C05558=1105.654,-74.562,-48.566,179.834,5.090,148.924
C05559=1105.648,-74.312,-48.578,179.834,5.095,148.925
C05560=1105.644,-74.063,-48.589,179.834,5.100,148.926
C05561=1105.639,-73.813,-48.600,179.834,5.105,148.927
C05562=1105.634,-73.563,-48.612,179.834,5.110,148.929
C05563=1105.629,-73.349,-48.622,179.834,5.114,148.929
C05564=1105.625,-73.135,-48.631,179.834,5.119,148.931
C05565=1105.620,-72.920,-48.641,179.833,5.123,148.932
C05566=1105.616,-72.706,-48.651,179.834,5.128,148.932
C05567=1105.611,-72.491,-48.660,179.833,5.132,148.933
C05568=1105.607,-72.276,-48.670,179.834,5.137,148.934
C05569=1105.602,-72.063,-48.679,179.833,5.141,148.936
C05570=1105.598,-71.848,-48.689,179.833,5.146,148.936
C05571=1105.593,-71.598,-48.701,179.833,5.151,148.938
C05572=1105.587,-71.349,-48.712,179.833,5.156,148.939
C05573=1105.582,-71.099,-48.724,179.834,5.161,148.940
C05574=1105.577,-70.849,-48.735,179.833,5.166,148.941
C05575=1105.571,-70.599,-48.747,179.833,5.171,148.942
C05576=1105.566,-70.350,-48.757,179.833,5.176,148.943
C05577=1105.561,-70.100,-48.769,179.833,5.181,148.944
C05578=1105.556,-69.850,-48.781,179.833,5.187,148.946
C05579=1105.551,-69.600,-48.793,179.833,5.191,148.947
C05580=1105.546,-69.351,-48.804,179.833,5.196,148.948
C05581=1105.540,-69.101,-48.816,179.833,5.202,148.949
C05582=1105.535,-68.852,-48.827,179.833,5.207,148.950
C05583=1105.530,-68.602,-48.839,179.833,5.212,148.951
C05584=1105.525,-68.352,-48.850,179.833,5.217,148.952
C05585=1105.520,-68.102,-48.862,179.833,5.222,148.953
C05586=1105.515,-67.853,-48.873,179.833,5.227,148.954
C05587=1105.509,-67.603,-48.885,179.833,5.232,148.956
C05588=1105.504,-67.354,-48.896,179.833,5.237,148.957
C05589=1105.499,-67.104,-48.908,179.833,5.242,148.958
C05590=1105.493,-66.854,-48.920,179.833,5.247,148.959
C05591=1105.489,-66.604,-48.931,179.833,5.252,148.960
C05592=1105.483,-66.354,-48.943,179.833,5.257,148.961
C05593=1105.479,-66.105,-48.954,179.833,5.262,148.962
C05594=1105.473,-65.855,-48.966,179.833,5.267,148.963
C05595=1105.468,-65.607,-48.978,179.833,5.272,148.964
C05596=1105.463,-65.357,-48.989,179.833,5.277,148.965
C05597=1105.457,-65.107,-49.001,179.833,5.282,148.966
C05598=1105.453,-64.857,-49.013,179.834,5.288,148.967
C05599=1105.447,-64.607,-49.024,179.834,5.293,148.969
C05600=1105.442,-64.358,-49.036,179.834,5.298,148.970
C05601=1105.437,-64.108,-49.048,179.834,5.303,148.971
C05602=1105.432,-63.858,-49.060,179.834,5.308,148.972
C05603=1105.427,-63.609,-49.072,179.834,5.313,148.973
C05604=1105.422,-63.359,-49.083,179.835,5.317,148.974
C05605=1105.416,-63.109,-49.095,179.835,5.323,148.975
C05606=1105.411,-62.860,-49.106,179.835,5.327,148.976
C05607=1105.406,-62.610,-49.118,179.835,5.332,148.977
C05608=1105.400,-62.361,-49.131,179.835,5.337,148.978
C05609=1105.396,-62.111,-49.142,179.835,5.342,148.979
C05610=1105.390,-61.861,-49.154,179.836,5.347,148.980
C05611=1105.385,-61.611,-49.166,179.835,5.352,148.981
C05612=1105.380,-61.361,-49.177,179.836,5.357,148.982
C05613=1105.375,-61.112,-49.190,179.836,5.362,148.983
C05614=1105.370,-60.862,-49.202,179.836,5.367,148.984
C05615=1105.364,-60.612,-49.213,179.837,5.372,148.985
C05616=1105.360,-60.363,-49.225,179.836,5.377,148.986
C05617=1105.354,-60.113,-49.237,179.837,5.381,148.987
C05618=1105.349,-59.863,-49.249,179.837,5.386,148.988
C05619=1105.345,-59.649,-49.260,179.837,5.390,148.989
C05620=1105.340,-59.435,-49.270,179.837,5.395,148.990
C05621=1105.336,-59.221,-49.280,179.837,5.399,148.991
C05622=1105.332,-59.006,-49.290,179.837,5.403,148.992
C05623=1105.327,-58.792,-49.301,179.837,5.407,148.993
C05624=1105.323,-58.578,-49.311,179.837,5.411,148.994
C05625=1105.319,-58.363,-49.321,179.836,5.415,148.995
C05626=1105.314,-58.148,-49.331,179.836,5.419,148.996
C05627=1105.309,-57.898,-49.343,179.837,5.423,148.997
C05628=1105.304,-57.649,-49.356,179.837,5.428,148.998
C05629=1105.298,-57.399,-49.368,179.836,5.432,148.999
C05630=1105.294,-57.150,-49.380,179.836,5.437,149.000
C05631=1105.289,-56.900,-49.392,179.836,5.443,149.001
C05632=1105.283,-56.650,-49.404,179.836,5.447,149.002
C05633=1105.278,-56.401,-49.416,179.836,5.452,149.003
C05634=1105.273,-56.151,-49.428,179.836,5.456,149.004
C05635=1105.268,-55.902,-49.440,179.836,5.461,149.005
C05636=1105.263,-55.652,-49.452,179.835,5.466,149.006
C05637=1105.257,-55.402,-49.464,179.836,5.471,149.007
C05638=1105.252,-55.153,-49.476,179.835,5.475,149.008
C05639=1105.247,-54.903,-49.488,179.835,5.480,149.009
C05640=1105.242,-54.654,-49.501,179.835,5.485,149.010
C05641=1105.236,-54.404,-49.513,179.835,5.489,149.012
C05642=1105.232,-54.155,-49.525,179.835,5.494,149.012
C05643=1105.226,-53.905,-49.537,179.835,5.499,149.014
C05644=1105.221,-53.655,-49.549,179.834,5.503,149.015
C05645=1105.216,-53.406,-49.561,179.835,5.508,149.016
C05646=1105.211,-53.156,-49.574,179.835,5.513,149.017
C05647=1105.206,-52.906,-49.586,179.834,5.518,149.018
C05648=1105.201,-52.656,-49.599,179.834,5.522,149.019
C05649=1105.195,-52.406,-49.611,179.834,5.527,149.020
C05650=1105.190,-52.157,-49.623,179.834,5.532,149.021
C05651=1105.185,-51.907,-49.635,179.834,5.536,149.022
C05652=1105.180,-51.658,-49.647,179.834,5.542,149.023
C05653=1105.175,-51.408,-49.659,179.833,5.546,149.024
C05654=1105.170,-51.159,-49.671,179.834,5.551,149.025
C05655=1105.165,-50.909,-49.684,179.834,5.556,149.027
C05656=1105.160,-50.659,-49.696,179.833,5.560,149.028
C05657=1105.155,-50.410,-49.709,179.833,5.565,149.029
C05658=1105.149,-50.160,-49.721,179.833,5.569,149.030
C05659=1105.144,-49.910,-49.733,179.833,5.574,149.031
C05660=1105.139,-49.661,-49.746,179.833,5.579,149.032
C05661=1105.134,-49.411,-49.758,179.832,5.583,149.033
C05662=1105.129,-49.162,-49.771,179.832,5.588,149.034
C05663=1105.123,-48.912,-49.782,179.832,5.594,149.035
C05664=1105.119,-48.662,-49.795,179.832,5.598,149.036
C05665=1105.113,-48.412,-49.808,179.832,5.603,149.037
C05666=1105.108,-48.162,-49.820,179.832,5.608,149.039
C05667=1105.103,-47.913,-49.832,179.832,5.612,149.039
C05668=1105.098,-47.664,-49.845,179.832,5.617,149.041
C05669=1105.092,-47.414,-49.857,179.832,5.622,149.042
C05670=1105.088,-47.164,-49.870,179.832,5.626,149.043
C05671=1105.083,-46.915,-49.882,179.831,5.631,149.044
C05672=1105.077,-46.665,-49.894,179.831,5.635,149.045
C05673=1105.072,-46.415,-49.907,179.831,5.640,149.046
C05674=1105.067,-46.166,-49.920,179.831,5.645,149.047
C05675=1105.062,-45.951,-49.931,179.831,5.649,149.048
C05676=1105.058,-45.737,-49.942,179.831,5.653,149.049
C05677=1105.054,-45.523,-49.952,179.830,5.657,149.050
C05678=1105.049,-45.309,-49.963,179.830,5.661,149.051
C05679=1105.044,-45.094,-49.973,179.830,5.665,149.052
C05680=1105.040,-44.880,-49.984,179.830,5.669,149.053
C05681=1105.036,-44.666,-49.995,179.829,5.673,149.054
C05682=1105.032,-44.451,-50.006,179.830,5.678,149.055
C05683=1105.027,-44.202,-50.019,179.829,5.682,149.056
C05684=1105.021,-43.953,-50.031,179.830,5.687,149.057
C05685=1105.016,-43.703,-50.043,179.829,5.691,149.058
C05686=1105.011,-43.453,-50.056,179.829,5.696,149.059
C05687=1105.006,-43.203,-50.069,179.829,5.702,149.060
C05688=1105.001,-42.954,-50.081,179.829,5.705,149.061
C05689=1104.996,-42.705,-50.094,179.829,5.711,149.062
C05690=1104.991,-42.454,-50.107,179.829,5.715,149.063
C05691=1104.985,-42.204,-50.119,179.829,5.720,149.064
C05692=1104.980,-41.955,-50.132,179.829,5.725,149.065
C05693=1104.975,-41.706,-50.145,179.829,5.730,149.066
C05694=1104.971,-41.456,-50.158,179.830,5.735,149.067
C05695=1104.965,-41.206,-50.170,179.830,5.740,149.068
C05696=1104.960,-40.957,-50.183,179.830,5.745,149.069
C05697=1104.955,-40.708,-50.196,179.831,5.750,149.070
C05698=1104.950,-40.457,-50.208,179.831,5.754,149.071
C05699=1104.945,-40.208,-50.221,179.831,5.758,149.072
C05700=1104.939,-39.958,-50.233,179.831,5.763,149.073
C05701=1104.934,-39.709,-50.247,179.831,5.768,149.074
C05702=1104.929,-39.459,-50.260,179.832,5.773,149.075
C05703=1104.924,-39.209,-50.272,179.832,5.778,149.076
C05704=1104.919,-38.960,-50.285,179.833,5.782,149.077
C05705=1104.914,-38.710,-50.298,179.833,5.786,149.078
C05706=1104.908,-38.460,-50.311,179.833,5.791,149.079
C05707=1104.903,-38.211,-50.323,179.833,5.796,149.080
C05708=1104.898,-37.962,-50.336,179.834,5.800,149.080
C05709=1104.894,-37.712,-50.349,179.834,5.804,149.081
C05710=1104.888,-37.462,-50.362,179.834,5.809,149.082
C05711=1104.883,-37.213,-50.375,179.835,5.814,149.083
C05712=1104.878,-36.963,-50.388,179.835,5.819,149.084
C05713=1104.873,-36.713,-50.400,179.835,5.823,149.085
C05714=1104.867,-36.464,-50.414,179.835,5.827,149.086
C05715=1104.863,-36.214,-50.427,179.836,5.832,149.087
C05716=1104.858,-35.964,-50.439,179.836,5.837,149.088
C05717=1104.852,-35.715,-50.452,179.836,5.841,149.089
C05718=1104.847,-35.465,-50.465,179.837,5.845,149.090
C05719=1104.842,-35.215,-50.478,179.837,5.850,149.090
C05720=1104.836,-34.966,-50.491,179.837,5.855,149.091
C05721=1104.832,-34.716,-50.505,179.837,5.859,149.092
C05722=1104.827,-34.467,-50.517,179.838,5.864,149.093
C05723=1104.822,-34.217,-50.531,179.838,5.868,149.094
C05724=1104.816,-33.967,-50.544,179.838,5.872,149.095
C05725=1104.811,-33.718,-50.556,179.838,5.877,149.096
C05726=1104.806,-33.468,-50.570,179.839,5.881,149.097
C05727=1104.801,-33.219,-50.582,179.839,5.885,149.098
C05728=1104.797,-32.969,-50.596,179.840,5.890,149.098
C05729=1104.791,-32.719,-50.609,179.840,5.895,149.099
C05730=1104.786,-32.470,-50.622,179.841,5.899,149.100
C05731=1104.781,-32.256,-50.633,179.841,5.903,149.101
C05732=1104.777,-32.041,-50.644,179.841,5.907,149.102
C05733=1104.772,-31.827,-50.656,179.841,5.910,149.103
C05734=1104.768,-31.613,-50.667,179.842,5.914,149.103
C05735=1104.764,-31.399,-50.678,179.841,5.918,149.104
C05736=1104.760,-31.185,-50.689,179.842,5.921,149.105
C05737=1104.755,-30.970,-50.701,179.843,5.926,149.105
C05738=1104.750,-30.756,-50.712,179.843,5.930,149.106
C05739=1104.746,-30.507,-50.725,179.842,5.934,149.107
C05740=1104.741,-30.257,-50.738,179.843,5.938,149.108
C05741=1104.735,-30.008,-50.751,179.843,5.943,149.109
C05742=1104.731,-29.758,-50.765,179.843,5.947,149.110
C05743=1104.725,-29.509,-50.778,179.844,5.952,149.111
C05744=1104.721,-29.259,-50.791,179.844,5.957,149.112
C05745=1104.715,-29.009,-50.805,179.845,5.961,149.113
C05746=1104.710,-28.760,-50.818,179.844,5.965,149.114
C05747=1104.705,-28.510,-50.831,179.845,5.970,149.115
C05748=1104.700,-28.260,-50.844,179.845,5.975,149.115
C05749=1104.695,-28.011,-50.858,179.845,5.979,149.116
C05750=1104.690,-27.761,-50.871,179.846,5.983,149.117
C05751=1104.685,-27.512,-50.884,179.846,5.988,149.118
C05752=1104.679,-27.263,-50.898,179.847,5.993,149.119
C05753=1104.675,-27.013,-50.911,179.847,5.997,149.120
C05754=1104.669,-26.763,-50.924,179.847,6.002,149.121
C05755=1104.665,-26.513,-50.938,179.847,6.007,149.122
C05756=1104.659,-26.263,-50.951,179.847,6.010,149.123
C05757=1104.655,-26.014,-50.964,179.847,6.015,149.124
C05758=1104.649,-25.764,-50.978,179.847,6.020,149.125
C05759=1104.644,-25.514,-50.991,179.848,6.025,149.126
C05760=1104.639,-25.265,-51.005,179.848,6.030,149.127
C05761=1104.633,-25.015,-51.018,179.848,6.034,149.128
C05762=1104.629,-24.766,-51.032,179.848,6.039,149.129
C05763=1104.623,-24.516,-51.045,179.849,6.044,149.130
C05764=1104.619,-24.267,-51.059,179.849,6.048,149.131
C05765=1104.613,-24.017,-51.072,179.850,6.053,149.132
C05766=1104.608,-23.768,-51.086,179.850,6.058,149.132
C05767=1104.603,-23.518,-51.099,179.849,6.062,149.134
C05768=1104.598,-23.269,-51.113,179.850,6.067,149.135
C05769=1104.593,-23.019,-51.126,179.850,6.071,149.135
C05770=1104.588,-22.770,-51.140,179.851,6.076,149.136
C05771=1104.582,-22.520,-51.153,179.851,6.081,149.137
C05772=1104.578,-22.271,-51.167,179.852,6.086,149.138
C05773=1104.573,-22.020,-51.180,179.852,6.090,149.139
C05774=1104.567,-21.771,-51.194,179.852,6.094,149.140
C05775=1104.563,-21.521,-51.207,179.852,6.099,149.141
C05776=1104.557,-21.272,-51.221,179.853,6.104,149.142
C05777=1104.553,-21.022,-51.234,179.853,6.109,149.143
C05778=1104.547,-20.773,-51.248,179.853,6.113,149.144
C05779=1104.542,-20.524,-51.262,179.853,6.118,149.145
C05780=1104.538,-20.273,-51.275,179.854,6.122,149.146
C05781=1104.532,-20.024,-51.289,179.854,6.127,149.146
C05782=1104.527,-19.774,-51.303,179.855,6.132,149.147
C05783=1104.521,-19.525,-51.317,179.855,6.136,149.148
C05784=1104.517,-19.276,-51.330,179.855,6.140,149.149
C05785=1104.512,-19.025,-51.344,179.856,6.145,149.150
C05786=1104.506,-18.776,-51.358,179.856,6.150,149.151
C05787=1104.503,-18.563,-51.369,179.857,6.153,149.152
C05788=1104.498,-18.348,-51.381,179.857,6.157,149.153
C05789=1104.494,-18.134,-51.393,179.857,6.162,149.153
C05790=1104.489,-17.920,-51.405,179.857,6.166,149.154
C05791=1104.485,-17.706,-51.417,179.858,6.169,149.155
C05792=1104.480,-17.491,-51.428,179.858,6.174,149.156
C05793=1104.476,-17.277,-51.440,179.859,6.177,149.156
C05794=1104.472,-17.064,-51.452,179.859,6.181,149.157
C05795=1104.467,-16.814,-51.466,179.859,6.186,149.158
C05796=1104.462,-16.564,-51.480,179.860,6.190,149.159
C05797=1104.456,-16.315,-51.494,179.860,6.195,149.160
C05798=1104.452,-16.065,-51.507,179.860,6.199,149.161
C05799=1104.447,-15.815,-51.521,179.861,6.204,149.162
C05800=1104.441,-15.566,-51.535,179.861,6.208,149.162
C05801=1104.436,-15.316,-51.549,179.862,6.213,149.163
C05802=1104.431,-15.066,-51.563,179.862,6.218,149.164
C05803=1104.426,-14.818,-51.577,179.862,6.222,149.165
C05804=1104.422,-14.568,-51.591,179.863,6.226,149.166
C05805=1104.416,-14.318,-51.604,179.864,6.231,149.167
C05806=1104.411,-14.069,-51.618,179.864,6.236,149.168
C05807=1104.406,-13.819,-51.633,179.865,6.240,149.169
C05808=1104.401,-13.569,-51.647,179.865,6.245,149.169
C05809=1104.397,-13.320,-51.661,179.865,6.249,149.170
C05810=1104.391,-13.071,-51.674,179.866,6.254,149.171
C05811=1104.386,-12.821,-51.689,179.867,6.258,149.172
C05812=1104.381,-12.571,-51.702,179.867,6.263,149.173
C05813=1104.376,-12.321,-51.717,179.868,6.267,149.174
C05814=1104.370,-12.072,-51.730,179.868,6.272,149.175
C05815=1104.365,-11.822,-51.745,179.868,6.276,149.176
C05816=1104.361,-11.573,-51.758,179.868,6.281,149.176
C05817=1104.356,-11.323,-51.773,179.869,6.285,149.177
C05818=1104.351,-11.074,-51.787,179.870,6.290,149.178
C05819=1104.346,-10.825,-51.801,179.870,6.295,149.179
C05820=1104.341,-10.575,-51.815,179.871,6.299,149.180
C05821=1104.336,-10.325,-51.829,179.871,6.303,149.181
C05822=1104.330,-10.076,-51.843,179.872,6.308,149.181
C05823=1104.325,-9.826,-51.858,179.872,6.312,149.182
C05824=1104.320,-9.577,-51.872,179.873,6.317,149.183
C05825=1104.315,-9.327,-51.886,179.873,6.322,149.184
C05826=1104.310,-9.077,-51.900,179.874,6.326,149.185
C05827=1104.305,-8.828,-51.914,179.874,6.330,149.186
C05828=1104.300,-8.579,-51.929,179.875,6.335,149.186
C05829=1104.296,-8.329,-51.942,179.875,6.339,149.187
C05830=1104.291,-8.079,-51.957,179.876,6.344,149.188
C05831=1104.286,-7.830,-51.971,179.877,6.348,149.189
C05832=1104.280,-7.581,-51.985,179.877,6.353,149.190
C05833=1104.275,-7.331,-51.999,179.878,6.358,149.191
C05834=1104.270,-7.081,-52.013,179.878,6.362,149.192
C05835=1104.265,-6.832,-52.028,179.879,6.366,149.192
C05836=1104.260,-6.582,-52.043,179.879,6.371,149.193
C05837=1104.254,-6.333,-52.056,179.880,6.376,149.194
C05838=1104.249,-6.083,-52.071,179.880,6.380,149.195
C05839=1104.244,-5.834,-52.086,179.881,6.385,149.196
C05840=1104.240,-5.584,-52.100,179.882,6.389,149.197
C05841=1104.235,-5.334,-52.114,179.882,6.394,149.197
C05842=1104.230,-5.085,-52.129,179.883,6.398,149.198
C05843=1104.225,-4.871,-52.141,179.883,6.402,149.199
C05844=1104.221,-4.657,-52.153,179.884,6.406,149.200
C05845=1104.217,-4.443,-52.166,179.884,6.409,149.200
C05846=1104.213,-4.229,-52.178,179.885,6.414,149.201
C05847=1104.208,-4.015,-52.190,179.885,6.417,149.202
C05848=1104.204,-3.801,-52.202,179.885,6.421,149.203
C05849=1104.199,-3.587,-52.216,179.886,6.425,149.203
C05850=1104.195,-3.373,-52.228,179.887,6.429,149.204
C05851=1104.190,-3.123,-52.242,179.887,6.434,149.205
C05852=1104.185,-2.873,-52.256,179.888,6.438,149.206
C05853=1104.180,-2.624,-52.271,179.889,6.443,149.206
C05854=1104.175,-2.375,-52.285,179.889,6.447,149.207
C05855=1104.170,-2.126,-52.299,179.890,6.452,149.208
C05856=1104.164,-1.875,-52.314,179.891,6.456,149.209
C05857=1104.160,-1.626,-52.329,179.891,6.460,149.210
C05858=1104.155,-1.377,-52.343,179.891,6.465,149.211
C05859=1104.150,-1.127,-52.358,179.892,6.469,149.211
C05860=1104.145,-0.878,-52.373,179.893,6.474,149.212
C05861=1104.140,-0.628,-52.387,179.893,6.479,149.213
C05862=1104.134,-0.378,-52.402,179.894,6.483,149.214
C05863=1104.130,-0.129,-52.417,179.895,6.488,149.215
C05864=1104.125,0.121,-52.431,179.895,6.493,149.216
C05865=1104.120,0.370,-52.445,179.896,6.497,149.216
C05866=1104.115,0.619,-52.460,179.897,6.502,149.217
C05867=1104.109,0.869,-52.475,179.897,6.506,149.218
C05868=1104.105,1.119,-52.490,179.898,6.511,149.219
C05869=1104.100,1.368,-52.505,179.899,6.515,149.220
C05870=1104.095,1.618,-52.519,179.899,6.520,149.220
C05871=1104.090,1.867,-52.534,179.900,6.525,149.221
C05872=1104.085,2.117,-52.549,179.900,6.529,149.222
C05873=1104.080,2.367,-52.563,179.901,6.533,149.223
C05874=1104.075,2.616,-52.578,179.901,6.538,149.224
C05875=1104.069,2.866,-52.593,179.902,6.542,149.225
C05876=1104.065,3.115,-52.608,179.903,6.547,149.225
C05877=1104.060,3.365,-52.622,179.903,6.552,149.226
C05878=1104.055,3.614,-52.637,179.904,6.556,149.227
C05879=1104.049,3.864,-52.652,179.904,6.561,149.228
C05880=1104.045,4.113,-52.667,179.905,6.565,149.229
C05881=1104.040,4.363,-52.681,179.906,6.570,149.230
C05882=1104.034,4.612,-52.697,179.907,6.575,149.230
C05883=1104.029,4.862,-52.711,179.908,6.579,149.231
C05884=1104.025,5.111,-52.726,179.908,6.584,149.232
C05885=1104.019,5.361,-52.741,179.909,6.588,149.233
C05886=1104.014,5.610,-52.756,179.909,6.593,149.234
C05887=1104.010,5.859,-52.771,179.910,6.597,149.234
C05888=1104.004,6.109,-52.786,179.911,6.602,149.235
C05889=1103.999,6.358,-52.801,179.911,6.607,149.236
C05890=1103.994,6.608,-52.815,179.912,6.612,149.237
C05891=1103.989,6.857,-52.831,179.913,6.616,149.238
C05892=1103.984,7.106,-52.846,179.913,6.621,149.239
C05893=1103.979,7.356,-52.861,179.915,6.626,149.240
C05894=1103.975,7.606,-52.876,179.915,6.631,149.240
C05895=1103.970,7.855,-52.891,179.916,6.635,149.241
C05896=1103.964,8.105,-52.906,179.917,6.640,149.242
C05897=1103.960,8.354,-52.921,179.917,6.645,149.243
C05898=1103.954,8.604,-52.936,179.918,6.649,149.244
C05899=1103.950,8.818,-52.948,179.918,6.653,149.244
C05900=1103.946,9.032,-52.961,179.918,6.657,149.245
C05901=1103.941,9.245,-52.975,179.918,6.660,149.246
C05902=1103.938,9.460,-52.987,179.918,6.664,149.247
C05903=1103.933,9.674,-53.001,179.919,6.668,149.248
C05904=1103.929,9.888,-53.014,179.920,6.672,149.248
C05905=1103.924,10.101,-53.027,179.920,6.676,149.249
C05906=1103.920,10.316,-53.039,179.920,6.679,149.250
C05907=1103.916,10.565,-53.054,179.921,6.684,149.251
C05908=1103.910,10.814,-53.070,179.921,6.688,149.252
C05909=1103.906,11.063,-53.085,179.921,6.693,149.252
C05910=1103.900,11.313,-53.100,179.922,6.697,149.253
C05911=1103.895,11.563,-53.115,179.922,6.701,149.254
C05912=1103.890,11.812,-53.130,179.922,6.706,149.255
C05913=1103.886,12.062,-53.146,179.923,6.711,149.256
C05914=1103.880,12.311,-53.161,179.923,6.715,149.257
C05915=1103.875,12.561,-53.176,179.923,6.719,149.258
C05916=1103.870,12.810,-53.191,179.924,6.724,149.258
C05917=1103.865,13.060,-53.207,179.924,6.728,149.259
C05918=1103.860,13.309,-53.222,179.925,6.732,149.260
C05919=1103.855,13.559,-53.238,179.925,6.737,149.261
C05920=1103.851,13.808,-53.253,179.925,6.741,149.262
C05921=1103.845,14.058,-53.268,179.926,6.746,149.263
C05922=1103.840,14.307,-53.283,179.927,6.750,149.264
C05923=1103.835,14.556,-53.298,179.927,6.754,149.264
C05924=1103.830,14.807,-53.314,179.927,6.759,149.265
C05925=1103.825,15.056,-53.329,179.928,6.763,149.266
C05926=1103.820,15.305,-53.345,179.928,6.767,149.267
C05927=1103.815,15.554,-53.360,179.929,6.771,149.268
C05928=1103.811,15.804,-53.376,179.930,6.776,149.269
C05929=1103.806,16.053,-53.391,179.930,6.780,149.270
C05930=1103.801,16.303,-53.406,179.930,6.785,149.270
C05931=1103.795,16.552,-53.422,179.931,6.789,149.271
C05932=1103.791,16.801,-53.437,179.931,6.793,149.272
C05933=1103.786,17.051,-53.453,179.932,6.798,149.273
C05934=1103.780,17.301,-53.468,179.933,6.802,149.274
C05935=1103.776,17.550,-53.483,179.933,6.806,149.274
C05936=1103.770,17.799,-53.499,179.933,6.811,149.275
C05937=1103.766,18.049,-53.515,179.934,6.815,149.276
C05938=1103.761,18.298,-53.530,179.934,6.819,149.277
C05939=1103.756,18.548,-53.546,179.935,6.824,149.278
C05940=1103.751,18.798,-53.561,179.935,6.828,149.279
C05941=1103.746,19.047,-53.576,179.936,6.832,149.279
C05942=1103.741,19.296,-53.592,179.936,6.836,149.280
C05943=1103.735,19.546,-53.608,179.937,6.841,149.281
C05944=1103.731,19.796,-53.623,179.937,6.845,149.282
C05945=1103.726,20.045,-53.639,179.938,6.849,149.283
C05946=1103.721,20.294,-53.654,179.939,6.854,149.283
C05947=1103.716,20.545,-53.670,179.939,6.858,149.284
C05948=1103.711,20.794,-53.685,179.940,6.862,149.285
C05949=1103.706,21.043,-53.701,179.940,6.867,149.286
C05950=1103.701,21.292,-53.717,179.941,6.870,149.286
C05951=1103.696,21.542,-53.733,179.941,6.875,149.287
C05952=1103.691,21.791,-53.748,179.942,6.880,149.288
C05953=1103.686,22.040,-53.764,179.942,6.883,149.289
C05954=1103.681,22.291,-53.780,179.943,6.888,149.290
C05955=1103.677,22.504,-53.792,179.944,6.891,149.290
C05956=1103.673,22.718,-53.807,179.944,6.895,149.291
C05957=1103.669,22.932,-53.820,179.944,6.898,149.292
C05958=1103.664,23.145,-53.833,179.945,6.903,149.292
C05959=1103.660,23.359,-53.847,179.946,6.906,149.293
C05960=1103.655,23.573,-53.860,179.946,6.910,149.294
C05961=1103.651,23.787,-53.874,179.947,6.913,149.294
C05962=1103.647,24.001,-53.887,179.947,6.917,149.295
C05963=1103.642,24.250,-53.903,179.948,6.921,149.296
C05964=1103.637,24.500,-53.919,179.949,6.925,149.296
C05965=1103.632,24.750,-53.935,179.949,6.929,149.297
C05966=1103.627,24.999,-53.950,179.950,6.934,149.298
C05967=1103.622,25.248,-53.966,179.950,6.937,149.299
C05968=1103.618,25.498,-53.982,179.951,6.942,149.299
C05969=1103.612,25.747,-53.998,179.952,6.946,149.300
C05970=1103.608,25.997,-54.014,179.952,6.950,149.301
C05971=1103.602,26.246,-54.030,179.953,6.954,149.302
C05972=1103.597,26.495,-54.046,179.954,6.959,149.302
C05973=1103.593,26.745,-54.062,179.954,6.963,149.303
C05974=1103.588,26.994,-54.077,179.955,6.967,149.304
C05975=1103.583,27.244,-54.093,179.956,6.972,149.305
C05976=1103.578,27.493,-54.109,179.956,6.975,149.305
C05977=1103.573,27.742,-54.125,179.957,6.979,149.306
C05978=1103.568,27.992,-54.141,179.958,6.984,149.307
C05979=1103.563,28.241,-54.157,179.958,6.988,149.307
C05980=1103.558,28.491,-54.173,179.960,6.992,149.308
C05981=1103.553,28.740,-54.190,179.960,6.997,149.309
C05982=1103.548,28.990,-54.205,179.961,7.000,149.310
C05983=1103.543,29.240,-54.221,179.962,7.004,149.310
C05984=1103.538,29.488,-54.237,179.962,7.009,149.311
C05985=1103.533,29.738,-54.253,179.963,7.013,149.312
C05986=1103.528,29.987,-54.270,179.964,7.017,149.313
C05987=1103.523,30.237,-54.286,179.965,7.021,149.313
C05988=1103.518,30.486,-54.302,179.965,7.025,149.314
C05989=1103.514,30.736,-54.317,179.966,7.029,149.315
C05990=1103.509,30.985,-54.334,179.967,7.034,149.315
C05991=1103.504,31.235,-54.350,179.967,7.037,149.316
C05992=1103.499,31.484,-54.366,179.968,7.042,149.317
C05993=1103.494,31.734,-54.382,179.969,7.046,149.318
C05994=1103.489,31.982,-54.398,179.969,7.050,149.318
C05995=1103.484,32.233,-54.414,179.970,7.054,149.319
C05996=1103.478,32.482,-54.431,179.972,7.058,149.320
C05997=1103.474,32.732,-54.447,179.972,7.062,149.320
C05998=1103.469,32.980,-54.463,179.973,7.067,149.321
C05999=1103.464,33.231,-54.479,179.974,7.071,149.322
C06000=1103.459,33.479,-54.495,179.974,7.074,149.322
C06001=1103.454,33.729,-54.511,179.975,7.079,149.323
C06002=1103.449,33.978,-54.528,179.976,7.083,149.324
C06003=1103.444,34.228,-54.544,179.977,7.087,149.324
C06004=1103.439,34.477,-54.560,179.977,7.091,149.325
C06005=1103.434,34.727,-54.577,179.978,7.096,149.326
C06006=1103.429,34.976,-54.592,179.979,7.099,149.327
C06007=1103.425,35.226,-54.609,179.980,7.103,149.327
C06008=1103.420,35.474,-54.625,179.981,7.108,149.328
C06009=1103.414,35.725,-54.642,179.981,7.111,149.329
C06010=1103.410,35.974,-54.658,179.982,7.115,149.329
C06011=1103.405,36.187,-54.672,179.983,7.119,149.330
C06012=1103.401,36.402,-54.686,179.984,7.122,149.330
C06013=1103.397,36.615,-54.701,179.984,7.126,149.331
C06014=1103.393,36.829,-54.714,179.985,7.129,149.332
C06015=1103.389,37.042,-54.728,179.986,7.133,149.332
C06016=1103.385,37.256,-54.742,179.987,7.137,149.333
C06017=1103.380,37.470,-54.756,179.987,7.140,149.333
C06018=1103.376,37.684,-54.770,179.988,7.143,149.334
C06019=1103.370,37.933,-54.787,179.989,7.148,149.334
C06020=1103.366,38.183,-54.804,179.990,7.151,149.335
C06021=1103.361,38.432,-54.819,179.991,7.155,149.336
C06022=1103.356,38.681,-54.836,179.992,7.160,149.336
C06023=1103.352,38.931,-54.853,179.992,7.163,149.337
C06024=1103.346,39.180,-54.870,179.993,7.167,149.338
C06025=1103.341,39.430,-54.886,179.994,7.172,149.338
C06026=1103.336,39.679,-54.902,179.995,7.176,149.339
C06027=1103.331,39.928,-54.919,179.996,7.180,149.340
C06028=1103.327,40.178,-54.935,179.997,7.184,149.340
C06029=1103.321,40.427,-54.952,179.998,7.188,149.341
C06030=1103.317,40.676,-54.969,179.998,7.192,149.342
C06031=1103.312,40.927,-54.985,179.999,7.196,149.342
C06032=1103.307,41.175,-55.001,-179.999,7.200,149.343
C06033=1103.302,41.425,-55.018,-179.999,7.204,149.344
C06034=1103.297,41.675,-55.035,-179.998,7.208,149.344
C06035=1103.292,41.923,-55.051,-179.997,7.212,149.345
C06036=1103.288,42.173,-55.068,-179.996,7.216,149.346
C06037=1103.282,42.423,-55.085,-179.995,7.220,149.346
C06038=1103.277,42.671,-55.102,-179.994,7.224,149.347
C06039=1103.273,42.921,-55.118,-179.993,7.228,149.347
C06040=1103.268,43.171,-55.136,-179.992,7.232,149.348
C06041=1103.262,43.419,-55.152,-179.991,7.236,149.349
C06042=1103.258,43.670,-55.168,-179.990,7.241,149.349
C06043=1103.252,43.919,-55.185,-179.990,7.244,149.350
C06044=1103.247,44.168,-55.201,-179.989,7.248,149.351
C06045=1103.243,44.418,-55.218,-179.987,7.253,149.351
C06046=1103.238,44.667,-55.235,-179.987,7.256,149.352
C06047=1103.233,44.917,-55.252,-179.985,7.260,149.352
C06048=1103.228,45.166,-55.268,-179.984,7.264,149.353
C06049=1103.223,45.416,-55.286,-179.984,7.268,149.354
C06050=1103.219,45.664,-55.303,-179.983,7.272,149.354
C06051=1103.214,45.913,-55.319,-179.982,7.277,149.355
C06052=1103.208,46.163,-55.336,-179.980,7.280,149.355
C06053=1103.204,46.412,-55.353,-179.980,7.284,149.356
C06054=1103.199,46.662,-55.370,-179.979,7.288,149.357
C06055=1103.194,46.911,-55.387,-179.978,7.293,149.357
C06056=1103.189,47.160,-55.403,-179.977,7.296,149.358
C06057=1103.184,47.410,-55.421,-179.976,7.300,149.359
C06058=1103.179,47.660,-55.437,-179.975,7.304,149.359
C06059=1103.174,47.910,-55.455,-179.974,7.308,149.360
C06060=1103.169,48.158,-55.471,-179.973,7.312,149.360
C06061=1103.164,48.408,-55.489,-179.971,7.316,149.361
C06062=1103.160,48.657,-55.506,-179.970,7.320,149.362
C06063=1103.155,48.906,-55.522,-179.970,7.324,149.362
C06064=1103.149,49.156,-55.539,-179.969,7.328,149.363
C06065=1103.145,49.405,-55.556,-179.967,7.332,149.363
C06066=1103.140,49.655,-55.573,-179.967,7.336,149.364
C06067=1103.136,49.868,-55.588,-179.965,7.339,149.364
C06068=1103.132,50.082,-55.603,-179.965,7.343,149.365
C06069=1103.127,50.296,-55.618,-179.964,7.346,149.366
C06070=1103.123,50.509,-55.632,-179.963,7.349,149.366
C06071=1103.119,50.723,-55.646,-179.962,7.353,149.367
C06072=1103.115,50.937,-55.661,-179.961,7.357,149.367
C06073=1103.111,51.151,-55.676,-179.960,7.360,149.367
C06074=1103.107,51.364,-55.690,-179.959,7.363,149.368
C06075=1103.102,51.613,-55.707,-179.958,7.367,149.369
C06076=1103.097,51.862,-55.725,-179.957,7.371,149.369
C06077=1103.091,52.112,-55.742,-179.956,7.375,149.370
C06078=1103.087,52.362,-55.759,-179.955,7.379,149.370
C06079=1103.082,52.611,-55.777,-179.954,7.383,149.371
C06080=1103.078,52.860,-55.793,-179.953,7.387,149.372
C06081=1103.072,53.109,-55.810,-179.952,7.391,149.372
C06082=1103.068,53.358,-55.827,-179.951,7.395,149.373
C06083=1103.062,53.608,-55.845,-179.950,7.399,149.373
C06084=1103.057,53.858,-55.862,-179.949,7.402,149.374
C06085=1103.053,54.107,-55.879,-179.947,7.407,149.374
C06086=1103.048,54.357,-55.897,-179.946,7.411,149.375
C06087=1103.044,54.605,-55.914,-179.945,7.415,149.376
C06088=1103.038,54.855,-55.931,-179.944,7.418,149.376
C06089=1103.033,55.104,-55.948,-179.943,7.422,149.377
C06090=1103.028,55.353,-55.966,-179.942,7.427,149.377
C06091=1103.023,55.603,-55.983,-179.941,7.431,149.378
C06092=1103.018,55.852,-56.001,-179.940,7.434,149.378
C06093=1103.014,56.102,-56.017,-179.939,7.438,149.379
C06094=1103.009,56.351,-56.035,-179.937,7.442,149.379
C06095=1103.004,56.601,-56.053,-179.936,7.446,149.380
C06096=1102.999,56.849,-56.070,-179.935,7.450,149.381
C06097=1102.994,57.099,-56.087,-179.934,7.454,149.381
C06098=1102.989,57.348,-56.105,-179.933,7.458,149.382
C06099=1102.985,57.598,-56.122,-179.931,7.462,149.382
C06100=1102.980,57.847,-56.140,-179.931,7.466,149.383
C06101=1102.975,58.097,-56.157,-179.929,7.469,149.383
C06102=1102.969,58.345,-56.175,-179.928,7.474,149.384
C06103=1102.965,58.595,-56.192,-179.927,7.478,149.384
C06104=1102.960,58.844,-56.210,-179.926,7.481,149.385
C06105=1102.955,59.094,-56.227,-179.925,7.485,149.386
C06106=1102.950,59.343,-56.245,-179.923,7.489,149.386
C06107=1102.946,59.592,-56.262,-179.922,7.494,149.387
C06108=1102.940,59.842,-56.279,-179.921,7.498,149.387
C06109=1102.935,60.091,-56.297,-179.920,7.501,149.388
C06110=1102.930,60.341,-56.315,-179.919,7.505,149.388
C06111=1102.926,60.589,-56.332,-179.918,7.509,149.389
C06112=1102.921,60.839,-56.350,-179.916,7.513,149.390
C06113=1102.916,61.088,-56.367,-179.916,7.517,149.390
C06114=1102.911,61.338,-56.385,-179.914,7.521,149.391
C06115=1102.906,61.587,-56.403,-179.913,7.525,149.391
C06116=1102.902,61.836,-56.420,-179.911,7.529,149.392
C06117=1102.897,62.085,-56.438,-179.910,7.533,149.392
C06118=1102.892,62.335,-56.456,-179.909,7.536,149.393
C06119=1102.887,62.584,-56.473,-179.908,7.540,149.393
C06120=1102.882,62.834,-56.492,-179.907,7.544,149.394
C06121=1102.877,63.084,-56.509,-179.905,7.548,149.394
C06122=1102.873,63.332,-56.527,-179.904,7.553,149.395
C06123=1102.868,63.572,-56.544,-179.903,7.556,149.395
C06124=1102.863,63.812,-56.561,-179.902,7.560,149.396
C06125=1102.858,64.052,-56.578,-179.901,7.563,149.396
C06126=1102.854,64.292,-56.596,-179.899,7.567,149.397
C06127=1102.850,64.532,-56.612,-179.898,7.571,149.398
C06128=1102.844,64.772,-56.629,-179.897,7.574,149.398
C06129=1102.840,65.012,-56.646,-179.896,7.578,149.398
C06130=1102.835,65.252,-56.664,-179.895,7.583,149.399
C06131=1102.831,65.501,-56.682,-179.893,7.587,149.400
C06132=1102.826,65.751,-56.699,-179.893,7.590,149.400
C06133=1102.821,66.000,-56.717,-179.891,7.594,149.401
C06134=1102.816,66.249,-56.735,-179.890,7.598,149.401
C06135=1102.811,66.498,-56.753,-179.888,7.602,149.402
C06136=1102.806,66.747,-56.771,-179.887,7.606,149.402
C06137=1102.802,66.997,-56.789,-179.886,7.610,149.403
C06138=1102.797,67.247,-56.807,-179.885,7.613,149.403
C06139=1102.792,67.496,-56.825,-179.883,7.617,149.404
C06140=1102.787,67.745,-56.843,-179.882,7.622,149.404
C06141=1102.782,67.995,-56.860,-179.881,7.625,149.405
C06142=1102.777,68.244,-56.878,-179.879,7.630,149.405
C06143=1102.772,68.493,-56.896,-179.878,7.634,149.406
C06144=1102.768,68.743,-56.915,-179.877,7.637,149.406
C06145=1102.763,68.992,-56.933,-179.876,7.641,149.407
C06146=1102.758,69.241,-56.951,-179.874,7.645,149.407
C06147=1102.753,69.490,-56.969,-179.873,7.649,149.408
C06148=1102.748,69.740,-56.987,-179.872,7.653,149.408
C06149=1102.743,69.989,-57.005,-179.870,7.657,149.409
C06150=1102.739,70.239,-57.023,-179.869,7.661,149.410
C06151=1102.734,70.488,-57.041,-179.868,7.664,149.410
C06152=1102.729,70.736,-57.060,-179.866,7.668,149.410
C06153=1102.724,70.986,-57.078,-179.865,7.673,149.411
C06154=1102.719,71.235,-57.096,-179.864,7.677,149.412
C06155=1102.714,71.484,-57.114,-179.862,7.680,149.412
C06156=1102.710,71.734,-57.133,-179.861,7.685,149.413
C06157=1102.705,71.983,-57.151,-179.860,7.688,149.413
C06158=1102.700,72.232,-57.168,-179.858,7.692,149.413
C06159=1102.695,72.482,-57.186,-179.857,7.696,149.414
C06160=1102.690,72.732,-57.205,-179.856,7.700,149.415
C06161=1102.686,72.980,-57.224,-179.854,7.704,149.415
C06162=1102.680,73.230,-57.242,-179.853,7.708,149.416
C06163=1102.453,63.273,-56.570,-179.900,7.553,149.394
C06164=1102.457,63.023,-56.552,-179.902,7.549,149.394
C06165=1102.462,62.773,-56.535,-179.903,7.545,149.393
C06166=1102.467,62.524,-56.517,-179.904,7.542,149.393
C06167=1102.472,62.275,-56.499,-179.905,7.538,149.392
C06168=1102.477,62.026,-56.481,-179.907,7.534,149.391
C06169=1102.482,61.776,-56.464,-179.908,7.530,149.391
C06170=1102.486,61.527,-56.446,-179.909,7.526,149.390
C06171=1102.491,61.278,-56.428,-179.910,7.523,149.390
C06172=1102.497,61.028,-56.411,-179.911,7.518,149.389
C06173=1102.501,60.779,-56.393,-179.913,7.514,149.389
C06174=1102.506,60.530,-56.375,-179.914,7.510,149.388
C06175=1102.511,60.281,-56.358,-179.915,7.507,149.388
C06176=1102.516,60.031,-56.340,-179.916,7.503,149.387
C06177=1102.521,59.782,-56.322,-179.917,7.498,149.386
C06178=1102.526,59.532,-56.305,-179.919,7.494,149.386
C06179=1102.530,59.284,-56.288,-179.920,7.490,149.385
C06180=1102.535,59.034,-56.271,-179.921,7.487,149.385
C06181=1102.540,58.785,-56.253,-179.922,7.483,149.384
C06182=1102.545,58.535,-56.235,-179.923,7.479,149.384
C06183=1102.550,58.286,-56.218,-179.924,7.475,149.383
C06184=1102.555,58.037,-56.200,-179.925,7.471,149.383
C06185=1102.560,57.787,-56.183,-179.926,7.467,149.382
C06186=1102.565,57.538,-56.165,-179.928,7.463,149.382
C06187=1102.569,57.288,-56.148,-179.929,7.459,149.381
C06188=1102.575,57.040,-56.130,-179.930,7.455,149.380
C06189=1102.580,56.790,-56.113,-179.931,7.452,149.380
C06190=1102.584,56.541,-56.096,-179.932,7.447,149.379
C06191=1102.589,56.291,-56.078,-179.934,7.443,149.379
C06192=1102.594,56.042,-56.061,-179.934,7.440,149.378
C06193=1102.599,55.793,-56.044,-179.936,7.436,149.378
C06194=1102.604,55.543,-56.026,-179.937,7.432,149.377
C06195=1102.609,55.294,-56.009,-179.938,7.427,149.376
C06196=1102.613,55.045,-55.991,-179.939,7.424,149.376
C06197=1102.618,54.795,-55.974,-179.940,7.420,149.375
C06198=1102.623,54.545,-55.957,-179.941,7.416,149.375
C06199=1102.628,54.296,-55.939,-179.943,7.412,149.374
C06200=1102.633,54.047,-55.922,-179.943,7.408,149.374
C06201=1102.638,53.798,-55.904,-179.945,7.404,149.373
C06202=1102.643,53.549,-55.888,-179.946,7.400,149.372
C06203=1102.648,53.299,-55.870,-179.947,7.396,149.372
C06204=1102.652,53.050,-55.853,-179.948,7.393,149.371
C06205=1102.657,52.800,-55.836,-179.949,7.388,149.371
C06206=1102.662,52.551,-55.819,-179.950,7.384,149.370
C06207=1102.667,52.301,-55.801,-179.951,7.381,149.370
C06208=1102.673,52.052,-55.784,-179.952,7.377,149.369
C06209=1102.677,51.803,-55.768,-179.953,7.372,149.368
C06210=1102.682,51.554,-55.750,-179.955,7.368,149.368
C06211=1102.686,51.304,-55.733,-179.955,7.365,149.367
C06212=1102.695,50.893,-55.704,-179.957,7.358,149.366
C06213=1102.702,50.483,-55.676,-179.959,7.351,149.365
C06214=1102.711,50.072,-55.648,-179.961,7.345,149.364
C06215=1102.719,49.660,-55.620,-179.962,7.338,149.363
C06216=1102.724,49.412,-55.603,-179.963,7.334,149.363
C06217=1102.729,49.162,-55.586,-179.964,7.331,149.362
C06218=1102.733,48.913,-55.569,-179.965,7.327,149.362
C06219=1102.739,48.663,-55.552,-179.966,7.322,149.361
C06220=1102.743,48.414,-55.535,-179.967,7.319,149.360
C06221=1102.749,48.165,-55.518,-179.968,7.315,149.360
C06222=1102.753,47.916,-55.501,-179.970,7.311,149.359
C06223=1102.758,47.666,-55.484,-179.971,7.306,149.359
C06224=1102.763,47.416,-55.467,-179.971,7.303,149.358
C06225=1102.768,47.166,-55.450,-179.972,7.298,149.357
C06226=1102.773,46.918,-55.434,-179.974,7.295,149.357
C06227=1102.777,46.668,-55.417,-179.974,7.291,149.356
C06228=1102.783,46.418,-55.400,-179.975,7.287,149.355
C06229=1102.787,46.169,-55.383,-179.976,7.282,149.355
C06230=1102.793,45.920,-55.365,-179.977,7.279,149.354
C06231=1102.797,45.671,-55.349,-179.978,7.275,149.354
C06232=1102.802,45.422,-55.332,-179.979,7.271,149.353
C06233=1102.807,45.172,-55.315,-179.981,7.266,149.352
C06234=1102.812,44.923,-55.299,-179.981,7.263,149.352
C06235=1102.816,44.673,-55.282,-179.982,7.259,149.351
C06236=1102.822,44.424,-55.265,-179.983,7.254,149.350
C06237=1102.827,44.175,-55.248,-179.984,7.251,149.350
C06238=1102.831,43.925,-55.232,-179.985,7.247,149.349
C06239=1102.836,43.676,-55.214,-179.986,7.243,149.349
C06240=1102.841,43.426,-55.198,-179.987,7.239,149.348
C06241=1102.846,43.177,-55.181,-179.988,7.235,149.347
C06242=1102.851,42.928,-55.164,-179.989,7.230,149.347
C06243=1102.856,42.678,-55.148,-179.989,7.227,149.346
C06244=1102.861,42.429,-55.131,-179.990,7.223,149.345
C06245=1102.866,42.179,-55.114,-179.991,7.218,149.345
C06246=1102.871,41.929,-55.098,-179.992,7.215,149.344
C06247=1102.876,41.681,-55.082,-179.993,7.211,149.344
C06248=1102.881,41.431,-55.064,-179.995,7.207,149.343
C06249=1102.886,41.181,-55.048,-179.996,7.202,149.342
C06250=1102.891,40.933,-55.031,-179.996,7.199,149.342
C06251=1102.895,40.683,-55.015,-179.997,7.195,149.341
C06252=1102.900,40.433,-54.998,-179.998,7.190,149.340
C06253=1102.905,40.184,-54.981,-179.999,7.187,149.340
C06254=1102.910,39.934,-54.965,-180.000,7.182,149.339
C06255=1102.915,39.685,-54.949,179.999,7.178,149.338
C06256=1102.920,39.436,-54.932,179.999,7.175,149.338
C06257=1102.925,39.186,-54.915,179.998,7.170,149.337
C06258=1102.930,38.938,-54.899,179.997,7.166,149.336
C06259=1102.935,38.688,-54.882,179.996,7.162,149.336
C06260=1102.939,38.438,-54.866,179.995,7.158,149.335
C06261=1102.945,38.189,-54.849,179.994,7.154,149.334
C06262=1102.950,37.939,-54.833,179.994,7.150,149.334
C06263=1102.955,37.691,-54.816,179.992,7.146,149.333
C06264=1102.959,37.476,-54.803,179.992,7.143,149.332
C06265=1102.963,37.263,-54.788,179.991,7.139,149.332
C06266=1102.967,37.049,-54.774,179.991,7.136,149.331
C06267=1102.972,36.835,-54.760,179.990,7.132,149.331
C06268=1102.976,36.622,-54.746,179.989,7.128,149.330
C06269=1102.980,36.408,-54.731,179.988,7.125,149.330
C06270=1102.984,36.194,-54.718,179.987,7.122,149.329
C06271=1102.989,35.981,-54.704,179.987,7.118,149.329
C06272=1102.993,35.731,-54.687,179.986,7.114,149.328
C06273=1102.998,35.481,-54.671,179.985,7.110,149.327
C06274=1103.003,35.232,-54.655,179.984,7.106,149.327
C06275=1103.008,34.983,-54.638,179.983,7.102,149.326
C06276=1103.013,34.733,-54.623,179.983,7.098,149.325
C06277=1103.018,34.483,-54.605,179.982,7.094,149.324
C06278=1103.024,34.234,-54.590,179.981,7.089,149.324
C06279=1103.028,33.985,-54.573,179.981,7.086,149.323
C06280=1103.033,33.736,-54.557,179.980,7.082,149.322
C06281=1103.038,33.486,-54.541,179.979,7.077,149.322
C06282=1103.043,33.237,-54.524,179.978,7.074,149.321
C06283=1103.048,32.987,-54.508,179.977,7.069,149.320
C06284=1103.053,32.738,-54.492,179.976,7.065,149.320
C06285=1103.057,32.489,-54.476,179.976,7.061,149.319
C06286=1103.063,32.239,-54.460,179.975,7.057,149.318
C06287=1103.067,31.990,-54.443,179.974,7.053,149.318
C06288=1103.073,31.740,-54.428,179.974,7.049,149.317
C06289=1103.077,31.491,-54.411,179.973,7.044,149.316
C06290=1103.082,31.241,-54.395,179.972,7.040,149.315
C06291=1103.087,30.992,-54.379,179.971,7.037,149.315
C06292=1103.092,30.742,-54.363,179.970,7.032,149.314
C06293=1103.097,30.493,-54.346,179.970,7.028,149.313
C06294=1103.102,30.244,-54.331,179.969,7.024,149.313
C06295=1103.107,29.994,-54.314,179.968,7.020,149.312
C06296=1103.112,29.745,-54.299,179.968,7.015,149.311
C06297=1103.117,29.495,-54.282,179.967,7.012,149.310
C06298=1103.122,29.246,-54.266,179.966,7.007,149.310
C06299=1103.126,28.996,-54.250,179.965,7.003,149.309
C06300=1103.132,28.747,-54.234,179.965,6.999,149.308
C06301=1103.137,28.497,-54.218,179.964,6.995,149.307
C06302=1103.142,28.248,-54.202,179.963,6.990,149.307
C06303=1103.147,27.999,-54.186,179.963,6.986,149.306
C06304=1103.151,27.749,-54.170,179.962,6.982,149.305
C06305=1103.157,27.500,-54.154,179.962,6.979,149.305
C06306=1103.161,27.250,-54.139,179.961,6.974,149.304
C06307=1103.166,27.001,-54.122,179.960,6.970,149.303
C06308=1103.171,26.751,-54.106,179.959,6.966,149.302
C06309=1103.176,26.502,-54.091,179.959,6.961,149.302
C06310=1103.181,26.253,-54.075,179.958,6.957,149.301
C06311=1103.186,26.003,-54.059,179.958,6.953,149.300
C06312=1103.191,25.753,-54.043,179.957,6.949,149.299
C06313=1103.196,25.504,-54.026,179.956,6.945,149.299
C06314=1103.201,25.254,-54.011,179.956,6.941,149.298
C06315=1103.206,25.005,-53.996,179.955,6.936,149.297
C06316=1103.210,24.756,-53.979,179.954,6.932,149.296
C06317=1103.216,24.507,-53.963,179.954,6.928,149.296
C06318=1103.221,24.256,-53.948,179.953,6.923,149.295
C06319=1103.226,24.007,-53.932,179.952,6.919,149.294
C06320=1103.230,23.794,-53.918,179.952,6.916,149.293
C06321=1103.234,23.580,-53.905,179.951,6.912,149.293
C06322=1103.238,23.366,-53.891,179.951,6.909,149.292
C06323=1103.243,23.152,-53.878,179.950,6.905,149.291
C06324=1103.247,22.938,-53.865,179.950,6.902,149.291
C06325=1103.251,22.725,-53.851,179.949,6.898,149.290
C06326=1103.256,22.511,-53.837,179.948,6.894,149.289
C06327=1103.259,22.297,-53.824,179.948,6.890,149.289
C06328=1103.265,22.047,-53.808,179.948,6.887,149.288
C06329=1103.270,21.798,-53.793,179.947,6.882,149.287
C06330=1103.275,21.548,-53.777,179.946,6.877,149.286
C06331=1103.279,21.299,-53.761,179.946,6.874,149.286
C06332=1103.285,21.050,-53.745,179.945,6.869,149.285
C06333=1103.289,20.800,-53.729,179.944,6.865,149.284
C06334=1103.295,20.550,-53.714,179.944,6.861,149.283
C06335=1103.299,20.301,-53.699,179.943,6.857,149.283
C06336=1103.304,20.051,-53.683,179.943,6.852,149.282
C06337=1103.310,19.802,-53.667,179.943,6.848,149.281
C06338=1103.314,19.553,-53.652,179.942,6.844,149.280
C06339=1103.320,19.303,-53.637,179.942,6.840,149.279
C06340=1103.324,19.054,-53.620,179.941,6.835,149.278
C06341=1103.330,18.804,-53.604,179.940,6.831,149.278
C06342=1103.334,18.555,-53.589,179.940,6.827,149.277
C06343=1103.339,18.305,-53.573,179.939,6.822,149.276
C06344=1103.344,18.056,-53.558,179.939,6.818,149.275
C06345=1103.349,17.807,-53.543,179.939,6.814,149.274
C06346=1103.354,17.557,-53.527,179.938,6.809,149.274
C06347=1103.359,17.307,-53.511,179.937,6.805,149.273
C06348=1103.364,17.058,-53.496,179.937,6.801,149.272
C06349=1103.369,16.809,-53.481,179.937,6.796,149.271
C06350=1103.375,16.559,-53.465,179.936,6.792,149.270
C06351=1103.379,16.310,-53.450,179.936,6.788,149.270
C06352=1103.384,16.060,-53.434,179.935,6.783,149.269
C06353=1103.389,15.811,-53.419,179.935,6.779,149.268
C06354=1103.394,15.562,-53.404,179.934,6.775,149.267
C06355=1103.399,15.312,-53.388,179.934,6.770,149.266
C06356=1103.403,15.062,-53.373,179.933,6.766,149.265
C06357=1103.409,14.813,-53.357,179.933,6.762,149.264
C06358=1103.415,14.563,-53.342,179.932,6.757,149.264
C06359=1103.419,14.314,-53.327,179.931,6.753,149.263
C06360=1103.424,14.064,-53.311,179.931,6.749,149.262
C06361=1103.429,13.815,-53.296,179.931,6.744,149.261
C06362=1103.434,13.565,-53.281,179.930,6.739,149.260
C06363=1103.439,13.316,-53.266,179.930,6.736,149.259
C06364=1103.444,13.067,-53.250,179.930,6.731,149.258
C06365=1103.448,12.817,-53.235,179.929,6.726,149.258
C06366=1103.453,12.568,-53.219,179.929,6.723,149.257
C06367=1103.459,12.318,-53.204,179.928,6.718,149.256
C06368=1103.464,12.069,-53.189,179.928,6.713,149.255
C06369=1103.469,11.819,-53.174,179.928,6.709,149.254
C06370=1103.473,11.569,-53.158,179.927,6.705,149.253
C06371=1103.479,11.320,-53.143,179.927,6.701,149.252
C06372=1103.484,11.070,-53.128,179.927,6.696,149.252
C06373=1103.489,10.821,-53.113,179.926,6.691,149.251
C06374=1103.494,10.572,-53.098,179.926,6.687,149.250
C06375=1103.499,10.322,-53.082,179.926,6.683,149.249
C06376=1103.503,10.108,-53.069,179.925,6.679,149.248
C06377=1103.508,9.894,-53.057,179.925,6.676,149.248
C06378=1103.511,9.680,-53.043,179.924,6.671,149.247
C06379=1103.516,9.467,-53.031,179.924,6.667,149.246
C06380=1103.520,9.252,-53.017,179.924,6.663,149.245
C06381=1103.524,9.039,-53.005,179.924,6.660,149.244
C06382=1103.529,8.825,-52.992,179.924,6.656,149.244
C06383=1103.533,8.611,-52.979,179.923,6.652,149.243
C06384=1103.538,8.361,-52.964,179.923,6.648,149.242
C06385=1103.543,8.112,-52.949,179.922,6.643,149.241
C06386=1103.548,7.863,-52.934,179.921,6.638,149.240
C06387=1103.553,7.613,-52.919,179.920,6.633,149.240
C06388=1103.558,7.364,-52.904,179.919,6.629,149.239
C06389=1103.563,7.114,-52.888,179.919,6.624,149.238
C06390=1103.568,6.864,-52.874,179.918,6.619,149.237
C06391=1103.572,6.615,-52.859,179.917,6.615,149.236
C06392=1103.578,6.365,-52.843,179.917,6.610,149.235
C06393=1103.583,6.116,-52.829,179.916,6.605,149.234
C06394=1103.588,5.866,-52.813,179.915,6.601,149.234
C06395=1103.593,5.617,-52.798,179.915,6.596,149.233
C06396=1103.598,5.367,-52.784,179.914,6.592,149.232
C06397=1103.603,5.118,-52.768,179.914,6.587,149.231
C06398=1103.608,4.868,-52.754,179.913,6.583,149.230
C06399=1103.613,4.619,-52.739,179.912,6.578,149.230
C06400=1103.618,4.369,-52.724,179.912,6.573,149.229
C06401=1103.623,4.120,-52.709,179.911,6.568,149.228
C06402=1103.628,3.870,-52.695,179.910,6.564,149.227
C06403=1103.633,3.621,-52.679,179.909,6.559,149.226
C06404=1103.638,3.371,-52.665,179.909,6.555,149.225
C06405=1103.643,3.122,-52.650,179.908,6.550,149.225
C06406=1103.648,2.872,-52.636,179.907,6.546,149.224
C06407=1103.653,2.623,-52.620,179.907,6.541,149.223
C06408=1103.658,2.373,-52.606,179.906,6.536,149.222
C06409=1103.663,2.124,-52.591,179.905,6.532,149.221
C06410=1103.669,1.874,-52.576,179.905,6.527,149.220
C06411=1103.673,1.625,-52.561,179.904,6.523,149.220
C06412=1103.678,1.375,-52.547,179.903,6.518,149.219
C06413=1103.683,1.126,-52.532,179.903,6.514,149.218
C06414=1103.689,0.876,-52.517,179.902,6.509,149.217
C06415=1103.694,0.627,-52.503,179.902,6.505,149.216
C06416=1103.698,0.378,-52.488,179.901,6.501,149.216
C06417=1103.703,0.128,-52.473,179.901,6.496,149.215
C06418=1103.708,-0.121,-52.458,179.900,6.491,149.214
C06419=1103.714,-0.371,-52.443,179.899,6.487,149.213
C06420=1103.718,-0.621,-52.429,179.899,6.482,149.212
C06421=1103.723,-0.870,-52.414,179.898,6.477,149.211
C06422=1103.728,-1.120,-52.400,179.898,6.473,149.210
C06423=1103.733,-1.370,-52.386,179.897,6.468,149.210
C06424=1103.738,-1.619,-52.370,179.896,6.464,149.209
C06425=1103.743,-1.869,-52.356,179.896,6.459,149.208
C06426=1103.748,-2.118,-52.341,179.895,6.455,149.207
C06427=1103.753,-2.368,-52.327,179.894,6.450,149.206
C06428=1103.758,-2.617,-52.312,179.894,6.446,149.205
C06429=1103.763,-2.867,-52.298,179.893,6.442,149.205
C06430=1103.768,-3.116,-52.284,179.893,6.437,149.204
C06431=1103.774,-3.366,-52.269,179.892,6.432,149.203
C06432=1103.778,-3.580,-52.256,179.892,6.429,149.202
C06433=1103.782,-3.794,-52.244,179.891,6.424,149.202
C06434=1103.787,-4.008,-52.232,179.890,6.421,149.201
C06435=1103.791,-4.221,-52.219,179.890,6.416,149.200
C06436=1103.795,-4.436,-52.207,179.889,6.413,149.199
C06437=1103.799,-4.650,-52.195,179.889,6.409,149.199
C06438=1103.804,-4.864,-52.182,179.889,6.405,149.198
C06439=1103.808,-5.078,-52.169,179.888,6.401,149.197
C06440=1103.813,-5.327,-52.155,179.887,6.396,149.197
C06441=1103.818,-5.577,-52.141,179.887,6.392,149.196
C06442=1103.823,-5.826,-52.127,179.887,6.388,149.195
C06443=1103.828,-6.076,-52.112,179.886,6.383,149.194
C06444=1103.833,-6.326,-52.098,179.885,6.379,149.193
C06445=1103.838,-6.575,-52.084,179.885,6.374,149.192
C06446=1103.843,-6.825,-52.069,179.884,6.369,149.191
C06447=1103.848,-7.074,-52.055,179.883,6.365,149.191
C06448=1103.853,-7.323,-52.041,179.883,6.360,149.190
C06449=1103.858,-7.573,-52.026,179.883,6.356,149.189
C06450=1103.863,-7.823,-52.012,179.882,6.352,149.188
C06451=1103.868,-8.072,-51.998,179.881,6.347,149.187
C06452=1103.874,-8.321,-51.984,179.881,6.343,149.186
C06453=1103.879,-8.571,-51.970,179.880,6.338,149.186
C06454=1103.884,-8.821,-51.955,179.880,6.333,149.185
C06455=1103.889,-9.071,-51.941,179.879,6.329,149.184
C06456=1103.894,-9.320,-51.927,179.879,6.325,149.183
C06457=1103.899,-9.570,-51.912,179.878,6.320,149.182
C06458=1103.904,-9.819,-51.899,179.878,6.315,149.181
C06459=1103.909,-10.069,-51.884,179.877,6.311,149.181
C06460=1103.914,-10.318,-51.870,179.876,6.306,149.180
C06461=1103.919,-10.568,-51.856,179.876,6.302,149.179
C06462=1103.925,-10.817,-51.842,179.876,6.298,149.178
C06463=1103.929,-11.067,-51.828,179.875,6.293,149.177
C06464=1103.934,-11.316,-51.814,179.874,6.289,149.176
C06465=1103.939,-11.566,-51.800,179.874,6.284,149.175
C06466=1103.944,-11.816,-51.785,179.873,6.279,149.175
C06467=1103.949,-12.065,-51.771,179.873,6.275,149.174
C06468=1103.954,-12.314,-51.757,179.873,6.271,149.173
C06469=1103.959,-12.564,-51.743,179.873,6.266,149.172
C06470=1103.964,-12.814,-51.729,179.872,6.262,149.171
C06471=1103.970,-13.063,-51.715,179.871,6.257,149.170
C06472=1103.975,-13.313,-51.701,179.871,6.252,149.169
C06473=1103.979,-13.563,-51.687,179.870,6.247,149.169
C06474=1103.985,-13.812,-51.673,179.870,6.244,149.168
C06475=1103.990,-14.061,-51.659,179.870,6.239,149.167
C06476=1103.995,-14.311,-51.645,179.869,6.234,149.166
C06477=1103.999,-14.561,-51.631,179.869,6.229,149.165
C06478=1104.005,-14.810,-51.617,179.868,6.225,149.164
C06479=1104.010,-15.060,-51.604,179.868,6.221,149.163
C06480=1104.015,-15.309,-51.589,179.867,6.216,149.162
C06481=1104.020,-15.558,-51.576,179.867,6.212,149.162
C06482=1104.025,-15.808,-51.561,179.866,6.207,149.161
C06483=1104.030,-16.058,-51.547,179.866,6.202,149.160
C06484=1104.035,-16.308,-51.534,179.865,6.197,149.159
C06485=1104.040,-16.557,-51.520,179.865,6.194,149.158
C06486=1104.045,-16.807,-51.506,179.865,6.189,149.157
C06487=1104.050,-17.056,-51.492,179.865,6.184,149.156
C06488=1104.055,-17.271,-51.480,179.864,6.181,149.155
C06489=1104.058,-17.484,-51.469,179.864,6.177,149.155
C06490=1104.063,-17.698,-51.457,179.863,6.172,149.154
C06491=1104.067,-17.912,-51.445,179.863,6.169,149.153
C06492=1104.072,-18.126,-51.433,179.863,6.165,149.152
C06493=1104.077,-18.341,-51.421,179.862,6.161,149.152
C06494=1104.081,-18.555,-51.409,179.862,6.157,149.151
C06495=1104.085,-18.768,-51.398,179.862,6.153,149.150
C06496=1104.090,-19.018,-51.384,179.861,6.148,149.149
C06497=1104.095,-19.268,-51.370,179.861,6.144,149.148
C06498=1104.101,-19.517,-51.356,179.860,6.139,149.147
C06499=1104.105,-19.767,-51.343,179.860,6.135,149.146
C06500=1104.111,-20.016,-51.329,179.860,6.130,149.146
C06501=1104.116,-20.266,-51.315,179.859,6.126,149.145
C06502=1104.120,-20.516,-51.302,179.859,6.121,149.144
C06503=1104.126,-20.765,-51.288,179.859,6.116,149.143
C06504=1104.131,-21.015,-51.274,179.859,6.112,149.142
C06505=1104.135,-21.265,-51.261,179.858,6.107,149.141
C06506=1104.141,-21.514,-51.247,179.858,6.102,149.140
C06507=1104.146,-21.764,-51.233,179.858,6.098,149.139
C06508=1104.151,-22.013,-51.220,179.857,6.093,149.138
C06509=1104.156,-22.263,-51.206,179.857,6.089,149.137
C06510=1104.162,-22.512,-51.193,179.857,6.084,149.136
C06511=1104.166,-22.762,-51.179,179.856,6.079,149.135
C06512=1104.171,-23.012,-51.165,179.856,6.075,149.134
C06513=1104.177,-23.261,-51.152,179.855,6.070,149.134
C06514=1104.181,-23.511,-51.139,179.856,6.066,149.132
C06515=1104.187,-23.760,-51.125,179.856,6.061,149.132
C06516=1104.191,-24.010,-51.112,179.855,6.056,149.131
C06517=1104.197,-24.259,-51.098,179.855,6.052,149.130
C06518=1104.202,-24.509,-51.084,179.854,6.047,149.129
C06519=1104.207,-24.758,-51.071,179.854,6.042,149.128
C06520=1104.212,-25.008,-51.057,179.854,6.038,149.127
C06521=1104.217,-25.257,-51.044,179.854,6.033,149.126
C06522=1104.222,-25.507,-51.030,179.853,6.028,149.125
C06523=1104.228,-25.757,-51.017,179.853,6.023,149.124
C06524=1104.232,-26.006,-51.004,179.853,6.018,149.123
C06525=1104.238,-26.257,-50.990,179.853,6.015,149.122
C06526=1104.242,-26.505,-50.977,179.853,6.010,149.121
C06527=1104.248,-26.756,-50.963,179.853,6.005,149.120
C06528=1104.252,-27.004,-50.950,179.852,6.000,149.119
C06529=1104.258,-27.255,-50.936,179.852,5.996,149.118
C06530=1104.263,-27.504,-50.924,179.852,5.991,149.117
C06531=1104.268,-27.754,-50.909,179.851,5.987,149.116
C06532=1104.273,-28.003,-50.897,179.851,5.982,149.115
C06533=1104.278,-28.254,-50.883,179.851,5.978,149.115
C06534=1104.283,-28.502,-50.870,179.850,5.973,149.114
C06535=1104.288,-28.753,-50.856,179.850,5.968,149.113
C06536=1104.293,-29.002,-50.844,179.850,5.964,149.112
C06537=1104.299,-29.251,-50.830,179.850,5.960,149.111
C06538=1104.303,-29.501,-50.817,179.849,5.955,149.110
C06539=1104.309,-29.750,-50.804,179.849,5.950,149.109
C06540=1104.314,-30.000,-50.790,179.849,5.946,149.108
C06541=1104.319,-30.249,-50.777,179.848,5.942,149.107
C06542=1104.324,-30.500,-50.764,179.848,5.937,149.106
C06543=1104.329,-30.749,-50.751,179.848,5.933,149.105
C06544=1104.334,-30.963,-50.739,179.847,5.929,149.105
C06545=1104.338,-31.177,-50.728,179.847,5.925,149.104
C06546=1104.342,-31.391,-50.716,179.847,5.921,149.103
C06547=1104.347,-31.606,-50.705,179.847,5.917,149.102
C06548=1104.351,-31.820,-50.694,179.847,5.914,149.102
C06549=1104.355,-32.034,-50.682,179.846,5.910,149.101
C06550=1104.359,-32.248,-50.672,179.846,5.905,149.100
C06551=1104.364,-32.462,-50.660,179.846,5.902,149.099
C06552=1104.369,-32.712,-50.648,179.846,5.898,149.098
C06553=1104.374,-32.961,-50.633,179.845,5.893,149.098
C06554=1104.379,-33.211,-50.621,179.845,5.889,149.097
C06555=1104.384,-33.460,-50.608,179.845,5.885,149.096
C06556=1104.390,-33.710,-50.595,179.844,5.880,149.095
C06557=1104.395,-33.960,-50.582,179.844,5.875,149.094
C06558=1104.399,-34.209,-50.568,179.844,5.872,149.093
C06559=1104.405,-34.459,-50.555,179.843,5.867,149.092
C06560=1104.410,-34.708,-50.543,179.843,5.862,149.091
C06561=1104.415,-34.958,-50.530,179.842,5.857,149.090
C06562=1104.420,-35.208,-50.516,179.843,5.853,149.090
C06563=1104.425,-35.458,-50.503,179.842,5.849,149.089
C06564=1104.430,-35.707,-50.491,179.842,5.844,149.088
C06565=1104.436,-35.957,-50.478,179.842,5.840,149.087
C06566=1104.440,-36.207,-50.465,179.841,5.835,149.086
C06567=1104.446,-36.456,-50.452,179.841,5.831,149.085
C06568=1104.451,-36.705,-50.438,179.840,5.826,149.084
C06569=1104.456,-36.955,-50.425,179.841,5.822,149.083
C06570=1104.461,-37.204,-50.413,179.840,5.817,149.082
C06571=1104.466,-37.454,-50.400,179.840,5.812,149.081
C06572=1104.471,-37.704,-50.386,179.839,5.808,149.080
C06573=1104.476,-37.953,-50.374,179.839,5.804,149.080
C06574=1104.481,-38.203,-50.361,179.839,5.799,149.079
C06575=1104.487,-38.453,-50.348,179.839,5.794,149.078
C06576=1104.492,-38.702,-50.335,179.838,5.790,149.077
C06577=1104.497,-38.952,-50.323,179.838,5.786,149.076
C06578=1104.501,-39.202,-50.310,179.838,5.781,149.075
C06579=1104.507,-39.451,-50.296,179.837,5.776,149.074
C06580=1104.512,-39.701,-50.284,179.837,5.771,149.073
C06581=1104.517,-39.950,-50.271,179.837,5.766,149.072
C06582=1104.522,-40.200,-50.258,179.837,5.762,149.071
C06583=1104.527,-40.450,-50.246,179.837,5.758,149.070
C06584=1104.533,-40.700,-50.233,179.836,5.753,149.069
C06585=1104.538,-40.950,-50.220,179.836,5.748,149.068
C06586=1104.543,-41.199,-50.208,179.836,5.743,149.067
C06587=1104.548,-41.448,-50.195,179.835,5.738,149.066
C06588=1104.553,-41.697,-50.182,179.835,5.733,149.065
C06589=1104.558,-41.948,-50.169,179.835,5.728,149.064
C06590=1104.564,-42.197,-50.156,179.835,5.723,149.063
C06591=1104.569,-42.446,-50.144,179.835,5.719,149.062
C06592=1104.574,-42.696,-50.132,179.835,5.714,149.061
C06593=1104.579,-42.946,-50.119,179.835,5.710,149.060
C06594=1104.584,-43.196,-50.106,179.835,5.704,149.059
C06595=1104.589,-43.445,-50.094,179.836,5.700,149.058
C06596=1104.594,-43.694,-50.081,179.835,5.695,149.057
C06597=1104.599,-43.945,-50.067,179.835,5.690,149.056
C06598=1104.605,-44.195,-50.055,179.836,5.686,149.055
C06599=1104.610,-44.444,-50.043,179.836,5.681,149.053
C06600=1104.614,-44.658,-50.032,179.836,5.677,149.053
C06601=1104.618,-44.872,-50.021,179.836,5.673,149.052
C06602=1104.623,-45.086,-50.010,179.836,5.669,149.051
C06603=1104.627,-45.301,-50.000,179.837,5.665,149.050
C06604=1104.631,-45.515,-49.989,179.837,5.661,149.049
C06605=1104.636,-45.729,-49.978,179.836,5.656,149.048
C06606=1104.640,-45.944,-49.967,179.837,5.652,149.047
C06607=1104.645,-46.157,-49.957,179.837,5.648,149.046
C06608=1104.650,-46.408,-49.944,179.837,5.644,149.045
C06609=1104.655,-46.657,-49.932,179.837,5.639,149.044
C06610=1104.660,-46.906,-49.919,179.837,5.634,149.043
C06611=1104.666,-47.156,-49.906,179.838,5.630,149.042
C06612=1104.671,-47.406,-49.894,179.838,5.625,149.041
C06613=1104.676,-47.656,-49.881,179.837,5.620,149.040
C06614=1104.681,-47.905,-49.869,179.838,5.616,149.038
C06615=1104.686,-48.155,-49.857,179.838,5.611,149.037
C06616=1104.691,-48.405,-49.844,179.839,5.606,149.036
C06617=1104.696,-48.654,-49.831,179.838,5.602,149.035
C06618=1104.702,-48.904,-49.820,179.838,5.596,149.034
C06619=1104.706,-49.154,-49.807,179.839,5.592,149.033
C06620=1104.712,-49.403,-49.794,179.839,5.587,149.032
C06621=1104.717,-49.653,-49.782,179.839,5.582,149.031
C06622=1104.722,-49.902,-49.770,179.839,5.578,149.030
C06623=1104.727,-50.152,-49.757,179.839,5.573,149.029
C06624=1104.733,-50.402,-49.745,179.839,5.568,149.028
C06625=1104.738,-50.651,-49.732,179.840,5.564,149.027
C06626=1104.743,-50.901,-49.721,179.839,5.559,149.026
C06627=1104.748,-51.151,-49.708,179.839,5.554,149.024
C06628=1104.753,-51.400,-49.695,179.840,5.550,149.023
C06629=1104.758,-51.650,-49.683,179.840,5.545,149.022
C06630=1104.763,-51.899,-49.671,179.840,5.540,149.021
C06631=1104.768,-52.149,-49.659,179.840,5.535,149.020
C06632=1104.773,-52.398,-49.647,179.840,5.531,149.019
C06633=1104.779,-52.648,-49.635,179.840,5.526,149.018
C06634=1104.784,-52.898,-49.622,179.841,5.521,149.017
C06635=1104.789,-53.148,-49.610,179.840,5.516,149.016
C06636=1104.794,-53.398,-49.597,179.841,5.512,149.015
C06637=1104.799,-53.647,-49.585,179.841,5.507,149.014
C06638=1104.804,-53.897,-49.573,179.841,5.502,149.013
C06639=1104.809,-54.146,-49.560,179.841,5.498,149.012
C06640=1104.815,-54.396,-49.548,179.841,5.493,149.010
C06641=1104.819,-54.645,-49.536,179.841,5.488,149.009
C06642=1104.825,-54.895,-49.524,179.842,5.484,149.008
C06643=1104.830,-55.145,-49.513,179.842,5.479,149.007
C06644=1104.835,-55.394,-49.500,179.841,5.474,149.006
C06645=1104.841,-55.644,-49.488,179.842,5.470,149.005
C06646=1104.846,-55.894,-49.475,179.842,5.465,149.004
C06647=1104.851,-56.143,-49.464,179.842,5.460,149.003
C06648=1104.856,-56.392,-49.452,179.842,5.455,149.002
C06649=1104.861,-56.642,-49.440,179.842,5.451,149.001
C06650=1104.866,-56.892,-49.427,179.842,5.446,149.000
C06651=1104.871,-57.142,-49.415,179.842,5.442,148.999
C06652=1104.876,-57.392,-49.403,179.842,5.436,148.998
C06653=1104.881,-57.641,-49.391,179.843,5.431,148.996
C06654=1104.886,-57.891,-49.379,179.843,5.427,148.996
C06655=1104.891,-58.141,-49.366,179.843,5.422,148.994
C06656=1104.896,-58.355,-49.357,179.843,5.418,148.993
C06657=1104.900,-58.569,-49.346,179.843,5.414,148.993
C06658=1104.905,-58.784,-49.336,179.843,5.410,148.992
C06659=1104.909,-58.997,-49.326,179.843,5.406,148.991
C06660=1104.914,-59.212,-49.316,179.843,5.402,148.990
C06661=1104.918,-59.427,-49.304,179.843,5.398,148.989
C06662=1104.923,-59.641,-49.295,179.843,5.394,148.988
C06663=1104.927,-59.855,-49.284,179.843,5.390,148.987
C06664=1104.932,-60.105,-49.273,179.843,5.385,148.986
C06665=1104.937,-60.355,-49.261,179.843,5.380,148.985
C06666=1104.943,-60.604,-49.248,179.843,5.376,148.984
C06667=1104.948,-60.854,-49.236,179.843,5.371,148.983
C06668=1104.953,-61.104,-49.225,179.842,5.366,148.982
C06669=1104.958,-61.353,-49.212,179.842,5.361,148.981
C06670=1104.963,-61.603,-49.201,179.842,5.356,148.980
C06671=1104.968,-61.853,-49.189,179.842,5.351,148.979
C06672=1104.973,-62.102,-49.177,179.842,5.346,148.978
C06673=1104.979,-62.352,-49.165,179.841,5.341,148.977
C06674=1104.984,-62.602,-49.153,179.841,5.335,148.976
C06675=1104.989,-62.851,-49.142,179.841,5.331,148.975
C06676=1104.994,-63.101,-49.130,179.841,5.325,148.974
C06677=1104.999,-63.351,-49.117,179.840,5.321,148.973
C06678=1105.004,-63.600,-49.106,179.840,5.316,148.972
C06679=1105.009,-63.850,-49.094,179.840,5.311,148.971
C06680=1105.015,-64.100,-49.082,179.840,5.306,148.970
C06681=1105.020,-64.349,-49.071,179.840,5.301,148.969
C06682=1105.025,-64.599,-49.059,179.840,5.296,148.967
C06683=1105.030,-64.848,-49.047,179.840,5.291,148.966
C06684=1105.035,-65.098,-49.035,179.840,5.286,148.965
C06685=1105.041,-65.348,-49.024,179.840,5.281,148.964
C06686=1105.045,-65.597,-49.012,179.840,5.276,148.963
C06687=1105.051,-65.847,-49.000,179.839,5.271,148.962
C06688=1105.056,-66.097,-48.988,179.840,5.266,148.961
C06689=1105.061,-66.347,-48.977,179.840,5.261,148.960
C06690=1105.066,-66.597,-48.965,179.839,5.256,148.959
C06691=1105.072,-66.846,-48.954,179.839,5.251,148.958
C06692=1105.077,-67.096,-48.942,179.840,5.246,148.957
C06693=1105.082,-67.345,-48.930,179.839,5.241,148.956
C06694=1105.087,-67.595,-48.919,179.839,5.236,148.954
C06695=1105.092,-67.845,-48.907,179.839,5.231,148.953
C06696=1105.097,-68.094,-48.895,179.840,5.225,148.952
C06697=1105.102,-68.344,-48.884,179.839,5.221,148.951
C06698=1105.108,-68.593,-48.873,179.839,5.216,148.950
C06699=1105.113,-68.843,-48.861,179.839,5.210,148.949
C06700=1105.118,-69.093,-48.849,179.840,5.205,148.948
C06701=1105.123,-69.343,-48.838,179.839,5.201,148.947
C06702=1105.128,-69.592,-48.826,179.839,5.195,148.946
C06703=1105.133,-69.842,-48.814,179.839,5.190,148.944
C06704=1105.139,-70.091,-48.803,179.840,5.185,148.943
C06705=1105.144,-70.341,-48.792,179.840,5.180,148.942
C06706=1105.150,-70.591,-48.780,179.840,5.175,148.941
C06707=1105.155,-70.841,-48.769,179.840,5.170,148.940
C06708=1105.160,-71.091,-48.757,179.840,5.165,148.939
C06709=1105.165,-71.340,-48.746,179.840,5.160,148.938
C06710=1105.170,-71.590,-48.735,179.840,5.155,148.936
C06711=1105.175,-71.840,-48.723,179.840,5.150,148.935
C06712=1105.180,-72.054,-48.713,179.840,5.145,148.934
C06713=1105.185,-72.269,-48.703,179.840,5.141,148.933
C06714=1105.188,-72.483,-48.694,179.840,5.136,148.932
C06715=1105.193,-72.697,-48.684,179.840,5.132,148.931
C06716=1105.197,-72.912,-48.674,179.840,5.127,148.930
C06717=1105.202,-73.126,-48.664,179.840,5.123,148.929
C06718=1105.207,-73.341,-48.654,179.840,5.118,148.928
C06719=1105.211,-73.554,-48.645,179.841,5.114,148.927
C06720=1105.216,-73.804,-48.633,179.841,5.109,148.926
C06721=1105.221,-74.055,-48.623,179.841,5.104,148.925
C06722=1105.227,-74.304,-48.611,179.841,5.099,148.924
C06723=1105.232,-74.553,-48.600,179.841,5.093,148.923
C06724=1105.237,-74.803,-48.588,179.841,5.088,148.921
C06725=1105.242,-75.053,-48.577,179.841,5.083,148.920
C06726=1105.248,-75.303,-48.566,179.842,5.078,148.919
C06727=1105.253,-75.553,-48.554,179.842,5.073,148.918
C06728=1105.258,-75.802,-48.543,179.842,5.068,148.917
C06729=1105.263,-76.051,-48.532,179.842,5.063,148.916
C06730=1105.269,-76.302,-48.521,179.842,5.057,148.914
C06731=1105.273,-76.551,-48.510,179.842,5.052,148.913
C06732=1105.279,-76.801,-48.498,179.842,5.047,148.912
C06733=1105.284,-77.050,-48.487,179.843,5.042,148.911
C06734=1105.289,-77.300,-48.476,179.843,5.037,148.910
C06735=1105.295,-77.550,-48.465,179.843,5.032,148.909
C06736=1105.300,-77.799,-48.454,179.843,5.027,148.907
C06737=1105.305,-78.049,-48.443,179.843,5.022,148.906
C06738=1105.310,-78.299,-48.431,179.843,5.016,148.905
C06739=1105.316,-78.548,-48.420,179.844,5.011,148.904
C06740=1105.321,-78.799,-48.410,179.844,5.006,148.903
C06741=1105.326,-79.049,-48.398,179.844,5.001,148.901
C06742=1105.331,-79.297,-48.387,179.844,4.996,148.900
C06743=1105.336,-79.548,-48.376,179.845,4.991,148.899
C06744=1105.341,-79.797,-48.365,179.845,4.986,148.898
C06745=1105.347,-80.047,-48.353,179.845,4.981,148.897
C06746=1105.352,-80.297,-48.343,179.845,4.976,148.896
C06747=1105.357,-80.546,-48.332,179.845,4.971,148.894
C06748=1105.362,-80.795,-48.321,179.846,4.965,148.893
C06749=1105.368,-81.046,-48.309,179.846,4.960,148.892
C06750=1105.372,-81.296,-48.298,179.846,4.955,148.891
C06751=1105.378,-81.545,-48.288,179.847,4.950,148.889
C06752=1105.383,-81.795,-48.277,179.847,4.945,148.888
C06753=1105.389,-82.045,-48.266,179.847,4.940,148.887
C06754=1105.394,-82.294,-48.255,179.847,4.935,148.886
C06755=1105.398,-82.544,-48.243,179.847,4.929,148.885
C06756=1105.404,-82.793,-48.233,179.848,4.925,148.884
C06757=1105.409,-83.043,-48.221,179.848,4.920,148.882
C06758=1105.414,-83.294,-48.211,179.849,4.914,148.881
C06759=1105.420,-83.542,-48.200,179.849,4.909,148.880
C06760=1105.425,-83.793,-48.189,179.849,4.904,148.879
C06761=1105.430,-84.042,-48.178,179.849,4.899,148.877
C06762=1105.435,-84.292,-48.168,179.850,4.894,148.876
C06763=1105.440,-84.542,-48.156,179.850,4.889,148.875
C06764=1105.446,-84.791,-48.146,179.850,4.884,148.874
C06765=1105.451,-85.041,-48.134,179.851,4.879,148.873
C06766=1105.456,-85.291,-48.124,179.851,4.874,148.872
C06767=1105.461,-85.540,-48.113,179.851,4.869,148.870
C06768=1105.466,-85.755,-48.104,179.852,4.865,148.869
C06769=1105.470,-85.969,-48.094,179.851,4.860,148.868
C06770=1105.475,-86.184,-48.085,179.852,4.856,148.867
C06771=1105.479,-86.398,-48.076,179.852,4.852,148.866
C06772=1105.484,-86.613,-48.066,179.852,4.847,148.865
C06773=1105.489,-86.827,-48.057,179.853,4.842,148.864
C06774=1105.493,-87.042,-48.048,179.853,4.839,148.863
C06775=1105.497,-87.256,-48.038,179.854,4.834,148.862
C06776=1105.503,-87.506,-48.028,179.854,4.829,148.861
C06777=1105.508,-87.756,-48.017,179.854,4.824,148.859
C06778=1105.513,-88.006,-48.006,179.854,4.819,148.858
C06779=1105.518,-88.255,-47.996,179.855,4.814,148.857
C06780=1105.523,-88.505,-47.985,179.855,4.809,148.856
C06781=1105.529,-88.755,-47.975,179.856,4.804,148.855
C06782=1105.534,-89.005,-47.964,179.856,4.799,148.854
C06783=1105.539,-89.254,-47.953,179.856,4.794,148.852
C06784=1105.544,-89.504,-47.943,179.856,4.789,148.851
C06785=1105.550,-89.754,-47.932,179.857,4.784,148.850
C06786=1105.554,-90.003,-47.921,179.858,4.779,148.849
C06787=1105.560,-90.253,-47.911,179.858,4.774,148.847
C06788=1105.565,-90.503,-47.900,179.858,4.769,148.846
C06789=1105.570,-90.752,-47.889,179.859,4.764,148.845
C06790=1105.576,-91.002,-47.878,179.859,4.759,148.844
C06791=1105.581,-91.252,-47.868,179.859,4.754,148.843
C06792=1105.586,-91.502,-47.857,179.859,4.749,148.841
C06793=1105.592,-91.751,-47.847,179.860,4.744,148.840
C06794=1105.597,-92.001,-47.836,179.860,4.739,148.839
C06795=1105.602,-92.251,-47.826,179.861,4.734,148.838
C06796=1105.607,-92.501,-47.814,179.861,4.730,148.837
C06797=1105.613,-92.750,-47.804,179.862,4.725,148.835
C06798=1105.618,-93.000,-47.794,179.862,4.720,148.834
C06799=1105.623,-93.250,-47.783,179.863,4.715,148.833
C06800=1105.627,-93.500,-47.774,179.863,4.710,148.832
C06801=1105.633,-93.749,-47.763,179.863,4.705,148.831
C06802=1105.638,-93.998,-47.752,179.864,4.700,148.829
C06803=1105.643,-94.249,-47.742,179.864,4.695,148.828
C06804=1105.649,-94.498,-47.732,179.865,4.690,148.827
C06805=1105.654,-94.748,-47.721,179.865,4.686,148.826
C06806=1105.659,-94.997,-47.710,179.866,4.680,148.824
C06807=1105.664,-95.247,-47.700,179.866,4.675,148.823
C06808=1105.670,-95.497,-47.689,179.866,4.670,148.822
C06809=1105.675,-95.747,-47.679,179.867,4.666,148.821
C06810=1105.680,-95.997,-47.669,179.867,4.661,148.820
C06811=1105.686,-96.246,-47.658,179.867,4.655,148.819
C06812=1105.691,-96.497,-47.648,179.868,4.651,148.817
C06813=1105.696,-96.746,-47.637,179.868,4.646,148.816
C06814=1105.701,-96.996,-47.626,179.869,4.641,148.815
C06815=1105.707,-97.245,-47.616,179.869,4.636,148.814
C06816=1105.712,-97.495,-47.606,179.870,4.631,148.813
C06817=1105.717,-97.745,-47.596,179.870,4.626,148.811
C06818=1105.722,-97.994,-47.586,179.871,4.622,148.810
C06819=1105.727,-98.245,-47.575,179.871,4.617,148.809
C06820=1105.733,-98.494,-47.565,179.871,4.612,148.808
C06821=1105.739,-98.744,-47.555,179.871,4.606,148.807
C06822=1105.744,-98.994,-47.544,179.872,4.602,148.805
C06823=1105.749,-99.243,-47.534,179.872,4.597,148.804
C06824=1105.753,-99.457,-47.525,179.872,4.593,148.803
C06825=1105.757,-99.672,-47.516,179.873,4.589,148.802
C06826=1105.763,-99.887,-47.507,179.873,4.584,148.801
C06827=1105.767,-100.101,-47.498,179.873,4.580,148.800
C06828=1105.771,-100.316,-47.490,179.874,4.576,148.799
C06829=1105.776,-100.531,-47.481,179.874,4.572,148.798
C06830=1105.780,-100.745,-47.472,179.875,4.568,148.797
C06831=1105.785,-100.959,-47.463,179.874,4.563,148.796
C06832=1105.790,-101.209,-47.453,179.875,4.559,148.795
C06833=1105.795,-101.459,-47.442,179.875,4.553,148.794
C06834=1105.801,-101.709,-47.432,179.876,4.548,148.792
C06835=1105.806,-101.958,-47.423,179.876,4.544,148.791
C06836=1105.811,-102.209,-47.413,179.877,4.539,148.790
C06837=1105.817,-102.458,-47.402,179.877,4.534,148.789
C06838=1105.822,-102.708,-47.392,179.877,4.528,148.788
C06839=1105.827,-102.958,-47.382,179.878,4.524,148.786
C06840=1105.832,-103.207,-47.372,179.879,4.519,148.785
C06841=1105.838,-103.457,-47.362,179.879,4.513,148.784
C06842=1105.843,-103.707,-47.351,179.879,4.508,148.783
C06843=1105.848,-103.957,-47.341,179.880,4.504,148.781
C06844=1105.853,-104.206,-47.331,179.880,4.499,148.780
C06845=1105.858,-104.456,-47.321,179.880,4.494,148.779
C06846=1105.864,-104.706,-47.311,179.881,4.488,148.778
C06847=1105.869,-104.955,-47.301,179.881,4.484,148.777
C06848=1105.874,-105.206,-47.291,179.882,4.479,148.775
C06849=1105.879,-105.455,-47.281,179.882,4.474,148.774
C06850=1105.885,-105.705,-47.271,179.882,4.469,148.773
C06851=1105.890,-105.954,-47.261,179.883,4.464,148.772
C06852=1105.895,-106.204,-47.251,179.883,4.459,148.771
C06853=1105.900,-106.454,-47.240,179.883,4.454,148.769
C06854=1105.905,-106.703,-47.231,179.884,4.449,148.768
C06855=1105.911,-106.954,-47.221,179.885,4.444,148.767
C06856=1105.916,-107.204,-47.211,179.885,4.439,148.766
C06857=1105.921,-107.453,-47.201,179.886,4.434,148.764
C06858=1105.927,-107.702,-47.191,179.886,4.429,148.763
C06859=1105.932,-107.953,-47.180,179.887,4.424,148.762
C06860=1105.937,-108.202,-47.171,179.887,4.419,148.761
C06861=1105.942,-108.452,-47.161,179.887,4.414,148.759
C06862=1105.948,-108.701,-47.151,179.887,4.409,148.758
C06863=1105.952,-108.951,-47.141,179.888,4.403,148.757
C06864=1105.958,-109.202,-47.132,179.889,4.399,148.756
C06865=1105.964,-109.451,-47.121,179.889,4.394,148.754
C06866=1105.969,-109.700,-47.112,179.889,4.389,148.753
C06867=1105.974,-109.950,-47.102,179.890,4.384,148.752
C06868=1105.980,-110.201,-47.092,179.890,4.378,148.751
C06869=1105.984,-110.450,-47.082,179.891,4.374,148.750
C06870=1105.990,-110.700,-47.072,179.891,4.369,148.748
C06871=1105.995,-110.949,-47.062,179.892,4.363,148.747
C06872=1106.000,-111.200,-47.052,179.892,4.358,148.746
C06873=1106.006,-111.449,-47.042,179.892,4.353,148.745
C06874=1106.011,-111.698,-47.033,179.893,4.349,148.743
C06875=1106.017,-111.949,-47.023,179.893,4.344,148.742
C06876=1106.021,-112.198,-47.013,179.894,4.338,148.741
C06877=1106.027,-112.447,-47.003,179.894,4.333,148.739
C06878=1106.032,-112.698,-46.994,179.895,4.328,148.738
C06879=1106.037,-112.947,-46.984,179.895,4.323,148.737
C06880=1106.042,-113.162,-46.975,179.895,4.319,148.736
C06881=1106.046,-113.376,-46.967,179.896,4.314,148.735
C06882=1106.051,-113.591,-46.959,179.896,4.310,148.734
C06883=1106.056,-113.806,-46.951,179.897,4.305,148.733
C06884=1106.061,-114.021,-46.942,179.897,4.301,148.732
C06885=1106.065,-114.236,-46.934,179.898,4.297,148.730
C06886=1106.069,-114.450,-46.925,179.898,4.292,148.730
C06887=1106.074,-114.665,-46.917,179.898,4.288,148.728
C06888=1106.079,-114.914,-46.907,179.899,4.283,148.727
C06889=1106.084,-115.164,-46.898,179.899,4.277,148.726
C06890=1106.089,-115.413,-46.888,179.900,4.273,148.725
C06891=1106.095,-115.664,-46.879,179.901,4.268,148.723
C06892=1106.100,-115.913,-46.869,179.901,4.262,148.722
C06893=1106.105,-116.164,-46.859,179.901,4.257,148.721
C06894=1106.110,-116.413,-46.850,179.901,4.252,148.720
C06895=1106.116,-116.663,-46.840,179.902,4.247,148.718
C06896=1106.121,-116.912,-46.830,179.902,4.241,148.717
C06897=1106.127,-117.162,-46.821,179.903,4.236,148.716
C06898=1106.132,-117.412,-46.811,179.904,4.232,148.714
C06899=1106.138,-117.662,-46.802,179.904,4.226,148.713
C06900=1106.143,-117.911,-46.792,179.905,4.221,148.712
C06901=1106.148,-118.161,-46.783,179.905,4.216,148.711
C06902=1106.153,-118.411,-46.773,179.906,4.211,148.709
C06903=1106.159,-118.661,-46.763,179.906,4.205,148.708
C06904=1106.163,-118.911,-46.754,179.906,4.200,148.707
C06905=1106.169,-119.160,-46.745,179.907,4.195,148.705
C06906=1106.174,-119.410,-46.735,179.907,4.190,148.704
C06907=1106.179,-119.660,-46.726,179.908,4.185,148.703
C06908=1106.185,-119.909,-46.715,179.908,4.180,148.702
C06909=1106.190,-120.159,-46.707,179.909,4.175,148.700
C06910=1106.196,-120.409,-46.697,179.910,4.169,148.699
C06911=1106.201,-120.659,-46.687,179.910,4.164,148.698
C06912=1106.206,-120.908,-46.679,179.911,4.159,148.696
C06913=1106.212,-121.158,-46.668,179.911,4.153,148.695
C06914=1106.217,-121.408,-46.659,179.912,4.148,148.694
C06915=1106.221,-121.658,-46.650,179.912,4.143,148.692
C06916=1106.227,-121.908,-46.640,179.912,4.138,148.691
C06917=1106.232,-122.158,-46.631,179.913,4.132,148.690
C06918=1106.237,-122.407,-46.621,179.913,4.127,148.688
C06919=1106.243,-122.657,-46.612,179.914,4.122,148.687
C06920=1106.248,-122.907,-46.603,179.915,4.116,148.686
C06921=1106.254,-123.157,-46.593,179.915,4.111,148.685
C06922=1106.259,-123.406,-46.584,179.916,4.106,148.683
C06923=1106.264,-123.656,-46.575,179.916,4.100,148.682
C06924=1106.269,-123.906,-46.565,179.917,4.096,148.680
C06925=1106.275,-124.156,-46.556,179.918,4.091,148.679
C06926=1106.280,-124.406,-46.547,179.918,4.085,148.678
C06927=1106.285,-124.655,-46.538,179.919,4.080,148.676
C06928=1106.291,-124.905,-46.528,179.919,4.075,148.675
C06929=1106.296,-125.155,-46.519,179.920,4.069,148.674
C06930=1106.301,-125.405,-46.510,179.920,4.064,148.673
C06931=1106.307,-125.655,-46.501,179.921,4.058,148.671
C06932=1106.312,-125.904,-46.491,179.921,4.053,148.670
C06933=1106.317,-126.154,-46.482,179.922,4.048,148.668
C06934=1106.322,-126.404,-46.473,179.922,4.043,148.667
C06935=1106.328,-126.654,-46.464,179.923,4.037,148.666
C06936=1106.333,-126.868,-46.455,179.923,4.032,148.665
C06937=1106.337,-127.083,-46.448,179.924,4.028,148.664
C06938=1106.341,-127.298,-46.440,179.924,4.023,148.662
C06939=1106.346,-127.513,-46.432,179.925,4.018,148.661
C06940=1106.350,-127.727,-46.424,179.925,4.014,148.660
C06941=1106.355,-127.942,-46.417,179.926,4.009,148.659
C06942=1106.360,-128.157,-46.408,179.926,4.004,148.658
C06943=1106.365,-128.372,-46.401,179.927,4.000,148.656
C06944=1105.941,-128.362,-46.427,179.934,4.004,148.655
C06945=1105.937,-128.147,-46.434,179.933,4.009,148.656
C06946=1105.932,-127.932,-46.442,179.933,4.014,148.657
C06947=1105.928,-127.718,-46.450,179.933,4.018,148.659
C06948=1105.923,-127.503,-46.458,179.932,4.022,148.660
C06949=1105.919,-127.288,-46.466,179.931,4.027,148.661
C06950=1105.914,-127.073,-46.474,179.931,4.031,148.662
C06951=1105.909,-126.859,-46.482,179.931,4.037,148.663
C06952=1105.905,-126.644,-46.489,179.930,4.041,148.664
C06953=1105.900,-126.395,-46.500,179.929,4.046,148.666
C06954=1105.894,-126.145,-46.508,179.929,4.052,148.667
C06955=1105.889,-125.895,-46.517,179.928,4.057,148.668
C06956=1105.883,-125.645,-46.527,179.928,4.062,148.670
C06957=1105.878,-125.395,-46.536,179.927,4.067,148.671
C06958=1105.873,-125.146,-46.545,179.926,4.073,148.673
C06959=1105.867,-124.895,-46.555,179.926,4.078,148.674
C06960=1105.862,-124.646,-46.564,179.925,4.084,148.675
C06961=1105.857,-124.396,-46.573,179.925,4.089,148.676
C06962=1105.851,-124.146,-46.583,179.924,4.094,148.678
C06963=1105.846,-123.896,-46.592,179.924,4.100,148.679
C06964=1105.841,-123.647,-46.601,179.923,4.105,148.681
C06965=1105.835,-123.397,-46.611,179.923,4.110,148.682
C06966=1105.831,-123.148,-46.621,179.923,4.115,148.683
C06967=1105.825,-122.898,-46.629,179.922,4.121,148.685
C06968=1105.820,-122.648,-46.639,179.921,4.126,148.686
C06969=1105.815,-122.398,-46.649,179.921,4.132,148.687
C06970=1105.810,-122.149,-46.657,179.920,4.137,148.688
C06971=1105.804,-121.898,-46.667,179.920,4.142,148.690
C06972=1105.799,-121.648,-46.677,179.919,4.147,148.691
C06973=1105.793,-121.398,-46.686,179.919,4.153,148.692
C06974=1105.789,-121.149,-46.696,179.918,4.157,148.694
C06975=1105.783,-120.899,-46.705,179.917,4.162,148.695
C06976=1105.778,-120.649,-46.714,179.917,4.168,148.696
C06977=1105.773,-120.400,-46.724,179.916,4.173,148.698
C06978=1105.767,-120.150,-46.733,179.916,4.178,148.699
C06979=1105.762,-119.900,-46.743,179.916,4.183,148.700
C06980=1105.757,-119.651,-46.752,179.915,4.189,148.702
C06981=1105.751,-119.401,-46.762,179.915,4.194,148.703
C06982=1105.746,-119.151,-46.771,179.914,4.199,148.704
C06983=1105.741,-118.901,-46.782,179.913,4.205,148.705
C06984=1105.736,-118.651,-46.791,179.913,4.210,148.707
C06985=1105.730,-118.402,-46.801,179.912,4.214,148.708
C06986=1105.725,-118.152,-46.810,179.912,4.220,148.709
C06987=1105.719,-117.902,-46.820,179.911,4.225,148.711
C06988=1105.714,-117.652,-46.829,179.911,4.230,148.712
C06989=1105.709,-117.403,-46.839,179.911,4.235,148.713
C06990=1105.704,-117.153,-46.848,179.910,4.241,148.714
C06991=1105.698,-116.903,-46.858,179.910,4.246,148.716
C06992=1105.693,-116.653,-46.867,179.909,4.251,148.717
C06993=1105.688,-116.403,-46.878,179.909,4.256,148.718
C06994=1105.683,-116.153,-46.886,179.908,4.261,148.720
C06995=1105.677,-115.904,-46.897,179.907,4.266,148.721
C06996=1105.672,-115.655,-46.906,179.907,4.271,148.722
C06997=1105.666,-115.405,-46.916,179.907,4.277,148.723
C06998=1105.661,-115.155,-46.925,179.906,4.282,148.725
C06999=1105.656,-114.904,-46.935,179.906,4.287,148.726
C07000=1105.651,-114.655,-46.945,179.905,4.292,148.727
C07001=1105.647,-114.441,-46.953,179.905,4.297,148.728
C07002=1105.642,-114.226,-46.962,179.904,4.301,148.729
C07003=1105.637,-114.011,-46.970,179.904,4.305,148.730
C07004=1105.632,-113.797,-46.979,179.904,4.310,148.731
C07005=1105.628,-113.583,-46.987,179.903,4.314,148.733
C07006=1105.623,-113.368,-46.995,179.903,4.318,148.734
C07007=1105.619,-113.153,-47.003,179.902,4.322,148.735
C07008=1105.615,-112.938,-47.012,179.902,4.327,148.736
C07009=1105.609,-112.688,-47.022,179.902,4.332,148.737
C07010=1105.604,-112.439,-47.032,179.901,4.337,148.738
C07011=1105.598,-112.189,-47.041,179.901,4.342,148.739
C07012=1105.593,-111.940,-47.051,179.900,4.347,148.741
C07013=1105.588,-111.689,-47.061,179.900,4.353,148.742
C07014=1105.583,-111.440,-47.071,179.900,4.358,148.743
C07015=1105.578,-111.190,-47.080,179.899,4.362,148.745
C07016=1105.572,-110.940,-47.091,179.898,4.367,148.746
C07017=1105.567,-110.691,-47.100,179.898,4.372,148.747
C07018=1105.562,-110.440,-47.110,179.897,4.378,148.748
C07019=1105.556,-110.191,-47.120,179.897,4.383,148.750
C07020=1105.552,-109.942,-47.130,179.896,4.387,148.751
C07021=1105.546,-109.692,-47.140,179.896,4.393,148.752
C07022=1105.541,-109.441,-47.150,179.896,4.398,148.753
C07023=1105.536,-109.192,-47.160,179.896,4.403,148.754
C07024=1105.530,-108.942,-47.170,179.895,4.408,148.756
C07025=1105.525,-108.693,-47.180,179.894,4.413,148.757
C07026=1105.520,-108.443,-47.190,179.894,4.418,148.758
C07027=1105.514,-108.193,-47.199,179.893,4.423,148.759
C07028=1105.509,-107.943,-47.210,179.893,4.428,148.761
C07029=1105.504,-107.694,-47.219,179.892,4.433,148.762
C07030=1105.499,-107.444,-47.230,179.892,4.438,148.763
C07031=1105.493,-107.194,-47.240,179.892,4.443,148.764
C07032=1105.488,-106.945,-47.250,179.892,4.448,148.765
C07033=1105.483,-106.694,-47.260,179.891,4.452,148.767
C07034=1105.478,-106.445,-47.270,179.890,4.458,148.768
C07035=1105.472,-106.195,-47.280,179.890,4.463,148.769
C07036=1105.467,-105.946,-47.290,179.890,4.468,148.771
C07037=1105.462,-105.696,-47.300,179.889,4.473,148.772
C07038=1105.457,-105.446,-47.310,179.889,4.478,148.773
C07039=1105.452,-105.197,-47.320,179.888,4.483,148.774
C07040=1105.447,-104.947,-47.331,179.888,4.488,148.775
C07041=1105.441,-104.696,-47.340,179.887,4.492,148.777
C07042=1105.435,-104.447,-47.350,179.887,4.497,148.778
C07043=1105.431,-104.197,-47.360,179.887,4.503,148.779
C07044=1105.425,-103.947,-47.370,179.887,4.508,148.780
C07045=1105.420,-103.698,-47.381,179.886,4.512,148.781
C07046=1105.415,-103.448,-47.391,179.886,4.517,148.783
C07047=1105.409,-103.198,-47.401,179.885,4.523,148.784
C07048=1105.404,-102.949,-47.411,179.885,4.528,148.785
C07049=1105.399,-102.699,-47.422,179.884,4.532,148.786
C07050=1105.394,-102.449,-47.432,179.884,4.537,148.788
C07051=1105.388,-102.199,-47.442,179.883,4.543,148.789
C07052=1105.384,-101.950,-47.452,179.883,4.548,148.790
C07053=1105.378,-101.700,-47.462,179.882,4.552,148.791
C07054=1105.373,-101.450,-47.472,179.882,4.557,148.792
C07055=1105.368,-101.200,-47.483,179.882,4.562,148.794
C07056=1105.362,-100.951,-47.493,179.881,4.567,148.795
C07057=1105.357,-100.736,-47.502,179.881,4.571,148.796
C07058=1105.354,-100.522,-47.511,179.881,4.576,148.797
C07059=1105.349,-100.307,-47.520,179.880,4.580,148.798
C07060=1105.344,-100.092,-47.528,179.880,4.584,148.799
C07061=1105.340,-99.878,-47.537,179.879,4.588,148.800
C07062=1105.335,-99.664,-47.546,179.879,4.593,148.801
C07063=1105.331,-99.449,-47.555,179.879,4.597,148.802
C07064=1105.326,-99.234,-47.563,179.879,4.601,148.803
C07065=1105.321,-98.985,-47.573,179.879,4.606,148.804
C07066=1105.316,-98.735,-47.585,179.877,4.611,148.806
C07067=1105.310,-98.485,-47.595,179.877,4.616,148.807
C07068=1105.305,-98.235,-47.605,179.877,4.621,148.808
C07069=1105.300,-97.986,-47.616,179.876,4.625,148.809
C07070=1105.294,-97.736,-47.626,179.876,4.630,148.810
C07071=1105.289,-97.486,-47.636,179.876,4.636,148.812
C07072=1105.284,-97.236,-47.647,179.875,4.641,148.813
C07073=1105.279,-96.986,-47.657,179.875,4.645,148.814
C07074=1105.274,-96.737,-47.667,179.874,4.650,148.815
C07075=1105.268,-96.488,-47.678,179.874,4.655,148.816
C07076=1105.263,-96.238,-47.688,179.873,4.660,148.818
C07077=1105.258,-95.988,-47.699,179.873,4.665,148.819
C07078=1105.253,-95.738,-47.709,179.873,4.670,148.820
C07079=1105.247,-95.488,-47.719,179.872,4.674,148.821
C07080=1105.242,-95.238,-47.730,179.872,4.679,148.822
C07081=1105.237,-94.989,-47.741,179.872,4.685,148.823
C07082=1105.231,-94.740,-47.751,179.871,4.689,148.825
C07083=1105.226,-94.489,-47.762,179.871,4.694,148.826
C07084=1105.221,-94.240,-47.772,179.871,4.699,148.827
C07085=1105.216,-93.990,-47.782,179.870,4.704,148.828
C07086=1105.210,-93.741,-47.793,179.870,4.709,148.829
C07087=1105.205,-93.490,-47.804,179.869,4.714,148.831
C07088=1105.200,-93.241,-47.814,179.869,4.719,148.832
C07089=1105.195,-92.991,-47.825,179.868,4.723,148.833
C07090=1105.190,-92.742,-47.836,179.868,4.728,148.834
C07091=1105.185,-92.491,-47.846,179.868,4.734,148.835
C07092=1105.179,-92.242,-47.856,179.867,4.738,148.837
C07093=1105.174,-91.992,-47.867,179.867,4.743,148.838
C07094=1105.169,-91.743,-47.878,179.867,4.748,148.839
C07095=1105.164,-91.492,-47.888,179.866,4.753,148.840
C07096=1105.158,-91.243,-47.899,179.866,4.758,148.841
C07097=1105.153,-90.993,-47.910,179.866,4.763,148.843
C07098=1105.148,-90.744,-47.920,179.865,4.768,148.844
C07099=1105.143,-90.494,-47.931,179.865,4.772,148.845
C07100=1105.138,-90.245,-47.942,179.864,4.777,148.846
C07101=1105.133,-89.994,-47.952,179.864,4.783,148.847
C07102=1105.127,-89.745,-47.962,179.864,4.788,148.849
C07103=1105.122,-89.495,-47.974,179.863,4.792,148.850
C07104=1105.117,-89.246,-47.984,179.863,4.798,148.851
C07105=1105.111,-88.995,-47.995,179.862,4.803,148.852
C07106=1105.106,-88.746,-48.006,179.862,4.808,148.853
C07107=1105.101,-88.496,-48.017,179.862,4.813,148.855
C07108=1105.095,-88.247,-48.028,179.861,4.817,148.856
C07109=1105.090,-87.997,-48.038,179.861,4.823,148.857
C07110=1105.085,-87.746,-48.049,179.861,4.828,148.858
C07111=1105.080,-87.498,-48.060,179.861,4.833,148.859
C07112=1105.075,-87.247,-48.070,179.861,4.838,148.861
C07113=1105.070,-87.033,-48.080,179.860,4.842,148.862
C07114=1105.066,-86.819,-48.089,179.860,4.846,148.863
C07115=1105.061,-86.604,-48.098,179.859,4.851,148.864
C07116=1105.057,-86.390,-48.107,179.859,4.855,148.865
C07117=1105.053,-86.175,-48.117,179.859,4.859,148.866
C07118=1105.047,-85.960,-48.126,179.858,4.864,148.867
C07119=1105.043,-85.747,-48.135,179.858,4.868,148.868
C07120=1105.039,-85.532,-48.145,179.858,4.873,148.869
C07121=1105.033,-85.282,-48.155,179.857,4.878,148.870
C07122=1105.029,-85.032,-48.167,179.857,4.883,148.871
C07123=1105.024,-84.782,-48.177,179.857,4.888,148.873
C07124=1105.018,-84.533,-48.188,179.856,4.892,148.874
C07125=1105.013,-84.283,-48.199,179.856,4.898,148.875
C07126=1105.007,-84.034,-48.210,179.856,4.903,148.876
C07127=1105.002,-83.784,-48.221,179.856,4.908,148.877
C07128=1104.998,-83.534,-48.232,179.856,4.913,148.879
C07129=1104.992,-83.284,-48.242,179.855,4.919,148.880
C07130=1104.987,-83.034,-48.254,179.855,4.924,148.881
C07131=1104.981,-82.786,-48.265,179.855,4.929,148.882
C07132=1104.976,-82.535,-48.276,179.854,4.934,148.884
C07133=1104.972,-82.286,-48.287,179.854,4.938,148.885
C07134=1104.966,-82.036,-48.297,179.854,4.943,148.886
C07135=1104.961,-81.786,-48.309,179.853,4.949,148.887
C07136=1104.956,-81.536,-48.320,179.853,4.954,148.888
C07137=1104.950,-81.287,-48.331,179.853,4.959,148.889
C07138=1104.946,-81.037,-48.342,179.853,4.964,148.891
C07139=1104.940,-80.787,-48.353,179.852,4.970,148.892
C07140=1104.935,-80.538,-48.364,179.852,4.975,148.893
C07141=1104.930,-80.288,-48.375,179.852,4.980,148.894
C07142=1104.924,-80.038,-48.386,179.852,4.985,148.896
C07143=1104.919,-79.789,-48.397,179.852,4.990,148.897
C07144=1104.914,-79.539,-48.409,179.851,4.995,148.898
C07145=1104.908,-79.289,-48.420,179.851,5.000,148.899
C07146=1104.903,-79.040,-48.431,179.851,5.006,148.900
C07147=1104.898,-78.790,-48.442,179.850,5.010,148.901
C07148=1104.893,-78.540,-48.453,179.850,5.015,148.903
C07149=1104.887,-78.291,-48.464,179.850,5.020,148.904
C07150=1104.883,-78.041,-48.475,179.850,5.025,148.905
C07151=1104.877,-77.790,-48.487,179.850,5.030,148.906
C07152=1104.872,-77.542,-48.498,179.850,5.036,148.907
C07153=1104.867,-77.292,-48.509,179.849,5.041,148.909
C07154=1104.862,-77.042,-48.521,179.849,5.046,148.910
C07155=1104.856,-76.792,-48.531,179.849,5.051,148.911
C07156=1104.851,-76.543,-48.542,179.849,5.056,148.912
C07157=1104.846,-76.293,-48.554,179.848,5.062,148.913
C07158=1104.841,-76.043,-48.565,179.848,5.067,148.915
C07159=1104.835,-75.793,-48.576,179.848,5.072,148.916
C07160=1104.830,-75.544,-48.587,179.848,5.077,148.917
C07161=1104.825,-75.294,-48.599,179.848,5.082,148.918
C07162=1104.820,-75.044,-48.611,179.848,5.087,148.919
C07163=1104.815,-74.795,-48.622,179.847,5.092,148.920
C07164=1104.809,-74.545,-48.633,179.848,5.097,148.921
C07165=1104.804,-74.295,-48.644,179.848,5.102,148.923
C07166=1104.800,-74.045,-48.655,179.847,5.107,148.924
C07167=1104.794,-73.796,-48.667,179.847,5.113,148.925
C07168=1104.789,-73.547,-48.678,179.847,5.118,148.926
C07169=1104.785,-73.332,-48.688,179.846,5.122,148.927
C07170=1104.780,-73.118,-48.698,179.847,5.127,148.928
C07171=1104.775,-72.903,-48.708,179.847,5.131,148.929
C07172=1104.770,-72.689,-48.717,179.847,5.136,148.930
C07173=1104.767,-72.474,-48.727,179.846,5.140,148.931
C07174=1104.762,-72.260,-48.737,179.847,5.145,148.932
C07175=1104.758,-72.046,-48.747,179.846,5.149,148.933
C07176=1104.753,-71.831,-48.757,179.847,5.153,148.934
C07177=1104.748,-71.582,-48.768,179.847,5.158,148.935
C07178=1104.743,-71.332,-48.780,179.846,5.164,148.936
C07179=1104.738,-71.082,-48.791,179.846,5.169,148.938
C07180=1104.732,-70.833,-48.803,179.846,5.174,148.939
C07181=1104.727,-70.583,-48.813,179.846,5.179,148.940
C07182=1104.722,-70.333,-48.825,179.846,5.184,148.941
C07183=1104.717,-70.083,-48.837,179.846,5.189,148.942
C07184=1104.711,-69.833,-48.848,179.846,5.194,148.943
C07185=1104.707,-69.584,-48.860,179.846,5.199,148.944
C07186=1104.701,-69.334,-48.871,179.846,5.204,148.946
C07187=1104.695,-69.084,-48.883,179.846,5.209,148.947
C07188=1104.691,-68.835,-48.894,179.846,5.214,148.948
C07189=1104.685,-68.586,-48.907,179.846,5.219,148.949
C07190=1104.681,-68.336,-48.918,179.846,5.224,148.950
C07191=1104.675,-68.086,-48.930,179.846,5.230,148.951
C07192=1104.671,-67.836,-48.941,179.846,5.234,148.952
C07193=1104.665,-67.587,-48.953,179.846,5.239,148.953
C07194=1104.659,-67.337,-48.965,179.846,5.245,148.954
C07195=1104.655,-67.088,-48.976,179.846,5.250,148.956
C07196=1104.649,-66.838,-48.988,179.846,5.254,148.957
C07197=1104.644,-66.588,-48.999,179.846,5.260,148.958
C07198=1104.639,-66.338,-49.011,179.846,5.265,148.959
C07199=1104.634,-66.088,-49.023,179.846,5.270,148.960
C07200=1104.629,-65.839,-49.034,179.846,5.275,148.961
C07201=1104.624,-65.589,-49.047,179.846,5.280,148.962
C07202=1104.618,-65.340,-49.058,179.846,5.285,148.963
C07203=1104.613,-65.090,-49.070,179.846,5.290,148.964
C07204=1104.608,-64.840,-49.082,179.846,5.295,148.965
C07205=1104.603,-64.591,-49.093,179.846,5.300,148.966
C07206=1104.597,-64.341,-49.105,179.846,5.305,148.967
C07207=1104.592,-64.092,-49.117,179.847,5.309,148.968
C07208=1104.588,-63.842,-49.129,179.847,5.315,148.970
C07209=1104.582,-63.592,-49.141,179.847,5.320,148.971
C07210=1104.577,-63.342,-49.153,179.847,5.324,148.972
C07211=1104.572,-63.092,-49.164,179.847,5.330,148.973
C07212=1104.567,-62.843,-49.176,179.847,5.334,148.974
C07213=1104.562,-62.593,-49.188,179.847,5.339,148.975
C07214=1104.556,-62.343,-49.200,179.847,5.344,148.976
C07215=1104.551,-62.094,-49.212,179.847,5.349,148.977
C07216=1104.546,-61.844,-49.224,179.848,5.354,148.978
C07217=1104.541,-61.594,-49.236,179.848,5.359,148.979
C07218=1104.536,-61.345,-49.247,179.848,5.364,148.980
C07219=1104.531,-61.095,-49.260,179.848,5.369,148.981
C07220=1104.526,-60.845,-49.272,179.848,5.374,148.982
C07221=1104.520,-60.595,-49.284,179.849,5.379,148.983
C07222=1104.516,-60.347,-49.296,179.849,5.384,148.984
C07223=1104.510,-60.097,-49.308,179.849,5.388,148.985
C07224=1104.505,-59.847,-49.319,179.849,5.393,148.986
C07225=1104.500,-59.633,-49.330,179.849,5.397,148.987
C07226=1104.496,-59.418,-49.340,179.849,5.401,148.988
C07227=1104.492,-59.204,-49.351,179.849,5.406,148.989
C07228=1104.487,-58.990,-49.360,179.849,5.410,148.990
C07229=1104.483,-58.776,-49.371,179.849,5.414,148.991
C07230=1104.479,-58.561,-49.382,179.849,5.418,148.992
C07231=1104.474,-58.347,-49.391,179.849,5.422,148.993
C07232=1104.469,-58.133,-49.403,179.848,5.426,148.993
C07233=1104.465,-57.883,-49.414,179.849,5.430,148.994
C07234=1104.459,-57.634,-49.426,179.849,5.435,148.996
C07235=1104.454,-57.384,-49.438,179.848,5.440,148.997
C07236=1104.449,-57.134,-49.450,179.848,5.444,148.998
C07237=1104.443,-56.885,-49.463,179.848,5.450,148.999
C07238=1104.439,-56.635,-49.474,179.848,5.454,149.000
C07239=1104.434,-56.386,-49.487,179.848,5.459,149.001
C07240=1104.429,-56.135,-49.499,179.848,5.464,149.002
C07241=1104.424,-55.886,-49.512,179.848,5.468,149.003
C07242=1104.418,-55.636,-49.523,179.848,5.473,149.004
C07243=1104.413,-55.386,-49.536,179.848,5.478,149.005
C07244=1104.408,-55.136,-49.548,179.847,5.482,149.006
C07245=1104.403,-54.887,-49.560,179.847,5.487,149.007
C07246=1104.398,-54.637,-49.572,179.848,5.492,149.008
C07247=1104.393,-54.388,-49.584,179.847,5.496,149.009
C07248=1104.387,-54.138,-49.596,179.847,5.501,149.011
C07249=1104.382,-53.889,-49.609,179.847,5.506,149.011
C07250=1104.377,-53.639,-49.621,179.847,5.510,149.013
C07251=1104.372,-53.390,-49.633,179.847,5.515,149.014
C07252=1104.367,-53.139,-49.646,179.847,5.520,149.015
C07253=1104.362,-52.890,-49.658,179.846,5.525,149.016
C07254=1104.356,-52.640,-49.670,179.847,5.529,149.017
C07255=1104.351,-52.390,-49.683,179.847,5.534,149.018
C07256=1104.346,-52.141,-49.695,179.846,5.539,149.019
C07257=1104.341,-51.891,-49.707,179.846,5.543,149.020
C07258=1104.335,-51.642,-49.720,179.846,5.549,149.021
C07259=1104.331,-51.392,-49.731,179.846,5.553,149.022
C07260=1104.326,-51.142,-49.744,179.846,5.558,149.023
C07261=1104.321,-50.893,-49.757,179.846,5.563,149.024
C07262=1104.316,-50.643,-49.769,179.845,5.567,149.026
C07263=1104.311,-50.394,-49.781,179.846,5.572,149.026
C07264=1104.305,-50.144,-49.794,179.846,5.577,149.028
C07265=1104.300,-49.894,-49.806,179.845,5.581,149.029
C07266=1104.295,-49.645,-49.818,179.845,5.586,149.030
C07267=1104.290,-49.394,-49.830,179.845,5.590,149.031
C07268=1104.285,-49.145,-49.843,179.845,5.595,149.032
C07269=1104.280,-48.896,-49.856,179.844,5.601,149.033
C07270=1104.274,-48.646,-49.869,179.844,5.605,149.034
C07271=1104.269,-48.396,-49.881,179.844,5.610,149.035
C07272=1104.263,-48.147,-49.893,179.844,5.615,149.036
C07273=1104.259,-47.897,-49.906,179.844,5.619,149.037
C07274=1104.253,-47.647,-49.918,179.844,5.624,149.038
C07275=1104.248,-47.398,-49.931,179.844,5.629,149.040
C07276=1104.243,-47.148,-49.943,179.843,5.633,149.041
C07277=1104.238,-46.899,-49.956,179.844,5.638,149.042
C07278=1104.233,-46.648,-49.968,179.844,5.643,149.043
C07279=1104.228,-46.399,-49.981,179.843,5.647,149.044
C07280=1104.223,-46.150,-49.993,179.843,5.652,149.045
C07281=1104.219,-45.936,-50.004,179.843,5.656,149.046
C07282=1104.214,-45.721,-50.016,179.843,5.660,149.047
C07283=1104.210,-45.507,-50.026,179.842,5.664,149.048
C07284=1104.206,-45.293,-50.037,179.842,5.668,149.049
C07285=1104.201,-45.079,-50.048,179.842,5.672,149.050
C07286=1104.197,-44.864,-50.059,179.842,5.677,149.051
C07287=1104.193,-44.650,-50.069,179.842,5.681,149.052
C07288=1104.187,-44.436,-50.080,179.842,5.685,149.052
C07289=1104.182,-44.186,-50.093,179.841,5.689,149.054
C07290=1104.177,-43.936,-50.105,179.842,5.694,149.055
C07291=1104.172,-43.687,-50.118,179.842,5.699,149.056
C07292=1104.167,-43.438,-50.130,179.841,5.703,149.057
C07293=1104.163,-43.188,-50.143,179.841,5.708,149.058
C07294=1104.157,-42.938,-50.156,179.841,5.712,149.059
C07295=1104.151,-42.688,-50.168,179.841,5.718,149.060
C07296=1104.146,-42.439,-50.181,179.841,5.723,149.061
C07297=1104.142,-42.189,-50.194,179.841,5.727,149.062
C07298=1104.137,-41.939,-50.207,179.842,5.732,149.063
C07299=1104.131,-41.690,-50.219,179.842,5.737,149.064
C07300=1104.126,-41.441,-50.232,179.842,5.742,149.065
C07301=1104.121,-41.191,-50.245,179.841,5.746,149.066
C07302=1104.116,-40.941,-50.258,179.842,5.751,149.067
C07303=1104.111,-40.692,-50.271,179.842,5.756,149.068
C07304=1104.106,-40.442,-50.283,179.842,5.761,149.069
C07305=1104.100,-40.192,-50.297,179.843,5.766,149.070
C07306=1104.095,-39.943,-50.309,179.843,5.770,149.071
C07307=1104.090,-39.694,-50.322,179.843,5.774,149.072
C07308=1104.086,-39.444,-50.335,179.843,5.779,149.073
C07309=1104.081,-39.194,-50.347,179.843,5.784,149.074
C07310=1104.075,-38.945,-50.361,179.844,5.789,149.075
C07311=1104.070,-38.695,-50.374,179.844,5.794,149.076
C07312=1104.065,-38.445,-50.386,179.844,5.798,149.077
C07313=1104.059,-38.196,-50.399,179.845,5.802,149.078
C07314=1104.055,-37.946,-50.412,179.845,5.807,149.079
C07315=1104.049,-37.696,-50.425,179.845,5.811,149.079
C07316=1104.044,-37.447,-50.438,179.845,5.816,149.080
C07317=1104.039,-37.197,-50.451,179.846,5.820,149.081
C07318=1104.034,-36.947,-50.464,179.846,5.825,149.082
C07319=1104.029,-36.698,-50.476,179.846,5.829,149.083
C07320=1104.024,-36.448,-50.490,179.846,5.834,149.084
C07321=1104.018,-36.198,-50.503,179.847,5.839,149.085
C07322=1104.013,-35.949,-50.515,179.847,5.843,149.086
C07323=1104.008,-35.699,-50.529,179.847,5.847,149.087
C07324=1104.003,-35.449,-50.541,179.848,5.852,149.088
C07325=1103.999,-35.200,-50.555,179.848,5.857,149.089
C07326=1103.993,-34.950,-50.568,179.848,5.861,149.090
C07327=1103.988,-34.701,-50.581,179.848,5.865,149.090
C07328=1103.983,-34.451,-50.594,179.849,5.870,149.091
C07329=1103.977,-34.201,-50.607,179.849,5.874,149.092
C07330=1103.972,-33.952,-50.620,179.849,5.879,149.093
C07331=1103.968,-33.703,-50.633,179.850,5.883,149.094
C07332=1103.962,-33.453,-50.646,179.850,5.887,149.095
C07333=1103.958,-33.203,-50.659,179.850,5.892,149.096
C07334=1103.952,-32.953,-50.673,179.851,5.897,149.097
C07335=1103.947,-32.703,-50.686,179.851,5.900,149.097
C07336=1103.942,-32.455,-50.699,179.851,5.905,149.098
C07337=1103.938,-32.240,-50.710,179.851,5.909,149.099
C07338=1103.934,-32.026,-50.721,179.851,5.913,149.100
C07339=1103.929,-31.812,-50.733,179.852,5.917,149.101
C07340=1103.924,-31.597,-50.744,179.853,5.921,149.101
C07341=1103.920,-31.383,-50.755,179.852,5.924,149.102
C07342=1103.916,-31.169,-50.767,179.853,5.928,149.103
C07343=1103.912,-30.955,-50.778,179.853,5.932,149.104
C07344=1103.907,-30.741,-50.790,179.853,5.936,149.105
C07345=1103.902,-30.492,-50.802,179.854,5.940,149.105
C07346=1103.896,-30.242,-50.816,179.854,5.945,149.106
C07347=1103.892,-29.993,-50.829,179.854,5.950,149.107
C07348=1103.886,-29.743,-50.842,179.854,5.954,149.108
C07349=1103.882,-29.493,-50.855,179.855,5.958,149.109
C07350=1103.876,-29.244,-50.869,179.855,5.963,149.110
C07351=1103.872,-28.994,-50.882,179.855,5.967,149.111
C07352=1103.866,-28.745,-50.895,179.856,5.972,149.112
C07353=1103.862,-28.495,-50.909,179.856,5.976,149.113
C07354=1103.856,-28.245,-50.922,179.856,5.981,149.114
C07355=1103.851,-27.995,-50.935,179.856,5.985,149.115
C07356=1103.846,-27.746,-50.949,179.857,5.990,149.115
C07357=1103.841,-27.496,-50.962,179.857,5.995,149.116
C07358=1103.835,-27.247,-50.975,179.858,5.999,149.117
C07359=1103.831,-26.997,-50.989,179.858,6.003,149.118
C07360=1103.825,-26.748,-51.002,179.858,6.008,149.119
C07361=1103.821,-26.498,-51.016,179.859,6.013,149.120
C07362=1103.815,-26.249,-51.029,179.859,6.018,149.121
C07363=1103.811,-25.999,-51.043,179.859,6.023,149.122
C07364=1103.806,-25.749,-51.056,179.859,6.026,149.123
C07365=1103.800,-25.500,-51.070,179.859,6.031,149.124
C07366=1103.796,-25.250,-51.083,179.859,6.036,149.125
C07367=1103.790,-25.000,-51.096,179.860,6.041,149.126
C07368=1103.786,-24.751,-51.110,179.860,6.046,149.127
C07369=1103.780,-24.501,-51.123,179.860,6.050,149.128
C07370=1103.775,-24.252,-51.137,179.860,6.055,149.129
C07371=1103.770,-24.002,-51.150,179.861,6.060,149.130
C07372=1103.765,-23.753,-51.164,179.861,6.064,149.131
C07373=1103.760,-23.503,-51.177,179.862,6.069,149.132
C07374=1103.755,-23.254,-51.191,179.861,6.073,149.132
C07375=1103.750,-23.004,-51.206,179.861,6.078,149.134
C07376=1103.745,-22.755,-51.218,179.862,6.083,149.134
C07377=1103.740,-22.505,-51.232,179.862,6.087,149.135
C07378=1103.734,-22.255,-51.246,179.863,6.092,149.136
C07379=1103.729,-22.006,-51.259,179.863,6.096,149.137
C07380=1103.724,-21.756,-51.273,179.863,6.101,149.138
C07381=1103.719,-21.506,-51.287,179.864,6.106,149.139
C07382=1103.714,-21.257,-51.301,179.864,6.110,149.140
C07383=1103.709,-21.007,-51.314,179.864,6.115,149.141
C07384=1103.704,-20.758,-51.328,179.865,6.120,149.142
C07385=1103.699,-20.508,-51.342,179.865,6.124,149.143
C07386=1103.694,-20.259,-51.355,179.865,6.129,149.144
C07387=1103.689,-20.009,-51.369,179.866,6.133,149.145
C07388=1103.683,-19.760,-51.382,179.866,6.138,149.146
C07389=1103.679,-19.510,-51.396,179.866,6.142,149.146
C07390=1103.674,-19.260,-51.410,179.866,6.147,149.147
C07391=1103.668,-19.011,-51.424,179.867,6.152,149.148
C07392=1103.663,-18.761,-51.437,179.867,6.156,149.149
C07393=1103.659,-18.547,-51.449,179.868,6.160,149.150
C07394=1103.655,-18.333,-51.461,179.868,6.164,149.151
C07395=1103.650,-18.119,-51.473,179.869,6.168,149.151
C07396=1103.645,-17.905,-51.485,179.868,6.172,149.152
C07397=1103.641,-17.691,-51.497,179.869,6.176,149.153
C07398=1103.638,-17.477,-51.508,179.869,6.180,149.154
C07399=1103.633,-17.263,-51.520,179.870,6.184,149.155
C07400=1103.629,-17.049,-51.532,179.870,6.187,149.155
C07401=1103.623,-16.800,-51.546,179.871,6.192,149.156
C07402=1103.618,-16.549,-51.560,179.871,6.197,149.157
C07403=1103.613,-16.300,-51.574,179.871,6.201,149.158
C07404=1103.608,-16.051,-51.588,179.871,6.205,149.159
C07405=1103.603,-15.801,-51.602,179.872,6.210,149.160
C07406=1103.598,-15.552,-51.616,179.872,6.215,149.161
C07407=1103.593,-15.301,-51.630,179.873,6.220,149.162
C07408=1103.588,-15.052,-51.644,179.873,6.224,149.162
C07409=1103.583,-14.803,-51.657,179.873,6.228,149.163
C07410=1103.578,-14.553,-51.672,179.874,6.233,149.164
C07411=1103.573,-14.304,-51.685,179.875,6.237,149.165
C07412=1103.568,-14.054,-51.700,179.875,6.242,149.166
C07413=1103.563,-13.804,-51.713,179.875,6.246,149.167
